// TwinCAT 3 PLC project SPS_Demo
// ProgramVersion: 3.1.4023.0
// libraries:
//   Tc2_ControllerToolbox, * (Beckhoff Automation GmbH)
//   Tc2_Math, * (Beckhoff Automation GmbH)
//   Tc2_MC2, * (Beckhoff Automation GmbH)
//   Tc2_MC2_Camming, * (Beckhoff Automation GmbH)
//   Tc2_Standard, * (Beckhoff Automation GmbH)
//   Tc2_System, * (Beckhoff Automation GmbH)
//   Tc2_Utilities, * (Beckhoff Automation GmbH)
//   Tc3_Module, * (Beckhoff Automation GmbH)
// project tree:
//   / AbwicklerTask.TcTTO, AufwicklerTask.TcTTO, DatenbearbeitungTask.TcTTO, FadenzugmotorTask.TcTTO, GlobalTextList.TcGTLO, MasterachseTask.TcTTO, PlcTask.TcTTO, Visualisierungsmanager.TcVMO (not stored)
//   DUTs/ DANCERCONTROL_ERRORS.TcDUT (not stored), DANCER_REF.TcDUT, E_DancerControlState.TcDUT (not stored), MoveState_t.TcDUT (not stored), MoveState_Fadenzugmotor.TcDUT (not stored), Regelungsmethode.TcDUT
//   GVLs/ GlobaleVariablen.TcGVL
//   POUs/Achsenzustandautom/ AbwicklerAnAus.TcPOU (not stored), AufwicklerAnAus.TcPOU, FadenzugmotorAnAus.TcPOU, MasterAnAus.TcPOU (not stored)
//   POUs/ MAIN.TcPOU
//   POUs/Regelungsmethode/ADRC-Regler/ ESO.TcPOU, Fal.TcPOU, TrackingDifferentiator.TcPOU, DiscreteTrackingDifferentiator.TcPOU, Sign.TcPOU
//   POUs/Regelungsmethode/IterativeLerningControl/ ILC.TcPOU, PRG_MovingAverage_1.TcPOU, Speicher_leeren.TcPOU
//   POUs/Regelungsmethode/KraftwerteBearbeiten/ Datenbearbeiten.TcPOU, PRG_Amplitudenbegrenzung.TcPOU, PRG_Analog2Volt.TcPOU, PRG_AntiPulsFilter.TcPOU, PRG_Durchschnitt.TcPOU, PRG_KalmannFilter.TcPOU, PRG_MovingAverage.TcPOU, PRG_Volt2Kraft.TcPOU
//   POUs/Regelungsmethode/PID-Regler/ PRG_PID_Abwickler.TcPOU, PRG_PID_Fadenzugmotor.TcPOU

CONFIGURATION SPS_Demo
    RESOURCE PLC ON TwinCAT3
        TASK AbwicklerTask(INTERVAL := T#100us, PRIORITY := 15);
        TASK AufwicklerTask(INTERVAL := T#100us, PRIORITY := 14);
        TASK DatenbearbeitungTask(INTERVAL := T#100us, PRIORITY := 2);
        TASK FadenzugmotorTask(INTERVAL := T#100us, PRIORITY := 3);
        TASK MasterachseTask(INTERVAL := T#100us, PRIORITY := 12);
        TASK PlcTask(INTERVAL := T#100us, PRIORITY := 1);
        PROGRAM AbwicklerAnAus WITH AbwicklerTask : AbwicklerAnAus;
        PROGRAM AufwicklerAnAus WITH AufwicklerTask : AufwicklerAnAus;
        PROGRAM Datenbearbeiten WITH DatenbearbeitungTask : Datenbearbeiten;
        PROGRAM Speicher_leeren WITH DatenbearbeitungTask : Speicher_leeren;
        PROGRAM FadenzugmotorAnAus WITH FadenzugmotorTask : FadenzugmotorAnAus;
        PROGRAM MasterAnAus WITH MasterachseTask : MasterAnAus;
        PROGRAM MAIN WITH PlcTask : MAIN;
    END_RESOURCE
END_CONFIGURATION

// ---- DUTs/DANCER_REF.TcDUT
TYPE DANCER_REF :
STRUCT
	/// 	Tension_ctl is the target value for web tension,
	///		typically the target position for the dancer in balanced condition 
	///	
	Tension_ctl: DINT;
	
	
	///	OUTPUT GearRatio
	///		GearRatio is the ratio of gear factor g(t)
	///		between master (web) and Slave (spool)
	///		to balance the dancer. Default is 1.0.
	///		GearRatio is an output value of the Dancercontrol function block.
	///	
	GearRatio: LREAL;
	
	
	
	/// 	deltaGear is the scaling multiplier of PID output (-1.0 ...  +1.0) to GearRatio - must be smaller than 1 but never 0.
	///		deltaGear would be e.g. 0.8 or 0.9 to limit the gear distortion 
	///		GearRatio = g(t) = deltaGear * PIDout + Gearoffset
	///	
	deltaGear: LREAL;
	
	
	
	/// 	GearOffset is the scaling offset to fit GearRatio distortion by satisfying equation
	///		GearRatio = g(t) = deltaGear * PIDout + Gearoffset
	///	
	GearOffset: LREAL;
	
	
	/// PID Control Proportional gain (P) 
	fKp: LREAL;
	
	
	/// PID Control Integral gain Tn (I) [s] 
	fTn: LREAL;
	
	
	/// PID Control Derivative gain Tv (D-T1) [s] 
	fTv: LREAL;
	
	
	/// PID Control Derivative damping time Td (D-T1) [s] 
	fTd: LREAL;
	
	
	/// 	acceleration limitation
	///		Accel_limit corresponds indirectly, i.e. relative to a
	///		maximum master velocity and to a maximum permitted 
	///		acceleration (pa = aSlaveMax / v MasterMax ). 
	///		The limit parameter pa corresponds to the 
	///		reciprocal value of the run-up time tH = 1 / pa 
	///	
	Accel_limit: LREAL;
END_STRUCT
END_TYPE

// ---- DUTs/Regelungsmethode.TcDUT
TYPE Regelungsmethode :
(
	Kraftkreis,
	On_Off
	
	
);
END_TYPE

// ---- GVLs/GlobaleVariablen.TcGVL
VAR_GLOBAL
	Master: 			AXIS_REF;
	Aufwickler: 		AXIS_REF;
	Abwickler: 			AXIS_REF;
	Fadenzugmotor		: AXIS_REF;		// Antrieb des Tänzers / Fadenzugausgleichssysmtems
	// Analog Input of EL3702 (Sample 0 ~ Sample 9 of Channel 1)
	aAnalogSamples_1 AT %I*: ARRAY[0..9] OF INT;
	// Analog Input of EL3702 (Sample 0 ~ Sample 9 of Channel 2)
	aAnalogSamples_2 AT %I*: ARRAY[0..9] OF INT;
	aAnalogSamplesReal_1: ARRAY[0..9] OF LREAL;
	aAnalogSamplesReal_2: ARRAY[0..9] OF LREAL;
	iAnalogSamplesAverageValue_1: LREAL := 0.36;
	iAnalogSamplesAverageValue_2: LREAL := 0.45;
	Reglerausgaenge: LREAL;
	ErrorTerm: LREAL;
	// Einheit (N)
	Sollkraft: LREAL := 10;
	Signal: LREAL;
	bPID_Regler_Switch: BOOL := FALSE;
	P_Regler_PseudoTorqCtrl_Out: LREAL;
	P_Regler_PTCVelocity_Out: LREAL;
	D_ReglerOut: LREAL;
	bI_Regler_Switch: BOOL := FALSE;
	bD_Regler_Switch: BOOL := FALSE;
	Fadenzugkraft_1: LREAL;
	Fadenzugkraft_2: LREAL;
	Sollposition: LREAL := 0;
	Istposition: LREAL;
	Stoerung: LREAL := 0;
	Stoerung_1: LREAL := 0;
	Stoerung_2: LREAL := 0;
	Positionsfehler: LREAL;
	KraftfehlerInPerzent: LREAL;
	stateAufwickler: Movestate_t;
	stateAbwickler: Movestate_t;
	xPunkt: LREAL := 360;
	MasterStart: BOOL;
	AufwicklerStart: BOOL;
	AbwicklerStart: BOOL;
	FadenmotorFreigabe: BOOL;
	MasterLaeuft: BOOL;
	AbwicklerLaeuft: BOOL;
	FadenzugHomingFertig: BOOL;
	FadenzugmotorLaeuft: BOOL;
	AufwicklerLaeuft: BOOL;
	Abwicklerstopp: BOOL;
	Aufwicklerstopp: BOOL;
	MasterStopp: BOOL;
	Straffunktion: LREAL;
	
	FadenmotorRegeln: BOOL:=FALSE;
	
	AbUndAufwicklersPosiabweichung: LREAL;
	AufwicklerJogStart: BOOL;
	FadenzugJogStart: BOOL;
	FadenzugmotorStopp: BOOL;
	NOT_AUS: BOOL;
	FadenzugmotorJogLaeuft: BOOL;
	AufwicklerJoglaeuft: BOOL;
	FadenzugmotorJogGes: LREAL;
	AufwicklerJogGes: LREAL;
	GearRatio: LREAL := 1;
	Regelungsmethode: STRING;
	v1: LREAL;
	v2: LREAL;
	ee:LREAL;//误差
	x1_hat:LREAL;//跟踪反馈值
	x2_hat:LREAL;//跟踪反馈值的而微分
	x3_hat:LREAL;//跟踪系统的扰动（总扰动）
	_u:LREAL;//输出值
	_u_neu: LREAL;
	u0:LREAL;//非线性组合系统输出
	
	ADRC_TD_r0:LREAL:=9000;
	ADRC_TD_h0:LREAL:=0.0001;
	// 3*wo
	ADRC_ESO_beta01:LREAL:=170;
	// 3*(wo^2)
	ADRC_ESO_beta02:LREAL:=5;
	// wo^3
	ADRC_ESO_beta03:LREAL:=0.01;
	b0:LREAL:=1.3;// 扰动补偿
	Referenzposition: LREAL := 90;
	ControlCycleTime: LREAL;
	P_Regler_Out_Abwickler: LREAL;
	I_Regler_Out_Abwickler: LREAL;
	I_Regler_Input_Abwickler: LREAL;
	D_Regler_Out_Abwickler: LREAL;
	PID_Output_After_Saturation_Abwickler: LREAL;
	//Kraftfehler: LREAL;
	PID_Output_After_Saturation_Fadenzugmotor: LREAL;
	Regler_Out_Fadenzugmotor: LREAL;
	P_Regler_Out_Fadenzugmotor: LREAL;
	I_Regler_Out_Fadenzugmotor: LREAL;
	D_Regler_Out_Fadenzugmotor: LREAL;
	I_Regler_Input_Fadenzugmotor: LREAL;
	// Grad
	MaxPosition: LREAL := 165;
	// Grad
	MinPosition: LREAL := 15;
	ADRC_Output:LREAL;
	KraftSensorNewValue: LREAL;
	KraftSensorOldValue: LREAL;
	Vorsteuerungsausgabe: LREAL;
	Kraftfehler: LREAL;
	KraftreglerOutput: LREAL;
	PID_Output_Old: ARRAY[0..20000] OF LREAL;
	ILC_Out: LREAL;
	k: INT := 2;
	Drehzahl: LREAL;
	u_new: LREAL;
	ILC_F_Out: LREAL;
	i:LREAL;
	LernenFertig: BOOL;
	ILC_EinAus:BOOL;
	neu_xPunkt: LREAL;
	alt_xPunkt: LREAL := xPunkt;
	xPunkt_geaendert: BOOL;
	u_Old: ARRAY[0..20000] OF LREAL;
	e_Old: ARRAY[0..20000] OF LREAL;
	count: INT;
	fla:BOOL:=FALSE;
	ADRC_ESO_h: LREAL := 0.0001;
	TD_Switch: BOOL;
	DTD_CTD: BOOL;
	E_Switch: BOOL;
END_VAR

// ---- POUs/Achsenzustandautom/AufwicklerAnAus.TcPOU
(* Ansteuerprogramm der Leitachse. Das Programm hat die Aufgabe, 
   die Leitachse in eine Bewegung konstanter Ge-schwindigkeit zu versetzen, 
   wieder anzuhalten und im Falle eines Fehlers die Achse durch einen Reset 
   wieder in einen funktionstüchtigen Zustand zu versetzen. *)

PROGRAM AufwicklerAnAus
VAR
	//stateMaster				: MoveState_t;		// Programmablauf über Zustandsvariable

	PowerAufwickler				: MC_Power;			// Schaltet Software-Freigabe der Leitachse
	HomeAufwicklerOut: ST_McOutputs;
	PowerAufwicklerOut			: ST_McOutputs;		// 
	
	ResetAufwickler				: MC_Reset;			// Setzt Achsfehler zurück
	ResetAufwicklerOut			: ST_McOutputs;	
	
	MoveAufwickler 				: MC_MoveVelocity;	// Versetzt Leitachse in Bewegung konstanter Geschwindigkeit
	MoveAufwicklerOut			: ST_McOutputs;
	
	HaltAufwickler				: MC_Halt;			// Hält Leitachse an
	GearInAufwicklerOut: ST_McOutputs;
	HaltAufwicklerOut			: ST_McOutputs;
	startAufwicklerTrig: R_TRIG;
	HaltAufwicklerTrig: R_TRIG;
	GearInAufwickler: MC_GearIn;
	GearOutAufwickler: MC_GearOut;
	CamOutAufwicklerOut: ST_McOutputs;
	CamInAufwicklerOut: ST_McOutputs;
	GearOutAufwicklerOut: ST_McOutputs;
	CamInAufwickler: MC_CamIn;
	CamOutAufwickler: MC_CamOut;
	SetCamOnlineChangeMode		: MC_SetCamOnlineChangeMode;				// Legt fest, wann und wie geänderte Kurvenscheibendaten übernommen werden
	SetCamOnlineChangeModeOut	: ST_McOutputs;
	
	CamTableSelect				: MC_CamTableSelect; // Spezifiziert und lädt Kurvenscheibentabelle in die NC
	
	MotionFunction				: ARRAY[1..4] OF MC_MotionFunctionPoint;	// Kurvenscheibe als Motion Function: Eindimensionale Liste (Array) von Stützstellen
	CamTable					: MC_CAM_REF;								// Referenz auf Kurvenscheibe: Beschreibung der Motion Function
	PointID						: MC_MotionFunctionPoint_ID;				// Wird den einzelnen Punkten/Stützstellen der Motion Function zugeordnet
	
	CamInfo						: MC_CamInfo;
	JogAufwicklerOut: ST_McOutputs;
	CamInfoOut					: ST_McOutputs;		
	CamInfoData					: MC_CamInfoData;	
	
	
	JogAufwickler: MC_Jog;
	flag: BOOL;
	AufwicklerHalt: MC_Halt;
	AufwicklerHaltOut: ST_McOutputs;
	HomeAufwickler: MC_Home;
	Kuppelungsmethode: BOOL;
	MARK: INT;
END_VAR

//startAufwicklerTrig(clk := MaschineStart);
//HaltAufwicklerTrig(clk := Abwicklerstopp);

GlobaleVariablen.Aufwickler();
CASE stateAufwickler OF
	
(* ===========================================================================================
   Zustand 1: Programm ist im Ausgangszustand und wartet auf Benutzereingabe. Alle 
   Funktionsbausteine werden initialisiert, etwaige Fehler zurückgesetzt. *)
	MOVESTATE_INIT :

		ResetAufwickler.Execute := FALSE;
		HaltAufwickler.Execute := FALSE;
		PowerAufwickler.Enable := FALSE;
		CamTableSelect.Execute := FALSE;
		CamInAufwickler.Execute := FALSE;
		CamOutAufwickler.Execute := FALSE;
		IF PowerAufwicklerOut.Active THEN
			ResetAufwickler.Execute := TRUE;
			IF ResetAufwickler.Done THEN
				AufwicklerLaeuft := FALSE;
				stateAufwickler := MOVESTATE_INIT;
			END_IF
		END_IF
		//HaltSlave.Execute := FALSE;
		//WriteMotionFunctionPoint.Execute := FALSE;
		//SetCamOnlineChangeMode.ActivationMode := MC_CAMACTIVATION_NEXTCYCLE;
		//SetCamOnlineChangeMode.MasterScalingMode := MC_CAMSCALING_AUTOOFFSET;
		//SetCamOnlineChangeMode.SlaveScalingMode := MC_CAMSCALING_AUTOOFFSET;
		IF AufwicklerStart = TRUE AND MasterLaeuft = FALSE THEN
			stateAufwickler := MOVESTATE_ENABLE;
		ELSIF AufwicklerStart = TRUE AND MasterLaeuft = TRUE THEN
			MasterStopp := TRUE;
		END_IF

(* ===========================================================================================
   Zustand 2: Schlalten der allgemeinen Software-Freigabe, Vorschubfreigabe in positive Richtung
   durch MC_Power. Sobald Funktionsbaustein MC_Power die Betriebsbereitschaft der Achse signalisiert,
   Zustandsübergang in Forward*)
	MOVESTATE_ENABLE :
			PowerAufwickler.Enable := TRUE;
			IF PowerAufwicklerOut.Done THEN
				stateAufwickler := MOVESTATE_HOMING;
			ELSIF PowerAufwickler.Error THEN
				stateAufwickler := MOVESTATE_ERROR;
			END_IF
	MOVESTATE_HOMING:
		IF AufwicklerStart = TRUE AND AufwicklerStopp = FALSE THEN
			HomeAufwickler.Execute := TRUE;

			IF HomeAufwicklerOut.Done THEN
				HomeAufwickler.Execute := FALSE;
				stateAufwickler := MOVESTATE_WRITEMOTIONFUNCTION;
				
			ELSIF HomeAufwicklerOut.CommandAborted OR HomeAufwicklerOut.Error THEN
				stateAufwickler := MOVESTATE_ERROR;
			END_IF
		END_IF	
(* ===========================================================================================
   Zustand 7: Beschreiben der zwei eindimensionalen Arrays mit der Stützstellen der Motion Function. 
   *)	
	MOVESTATE_WRITEMOTIONFUNCTION :
		PointID := 1;												// Dient nur der richtigen Position im Array
			MotionFunction[PointID].PointIndex			:= 1;		// Index der Stützstelle innerhalb der Motion Function
			MotionFunction[PointID].FunctionType 		:= 23;		// Modifizierte Sinuslinie
			MotionFunction[PointID].PointType    		:= 16#0002; // Motion Point Type : Rastpunkt
			MotionFunction[PointID].RelIndexNextPoint 	:= 1;		// Angabe des nächsten Punktes
			MotionFunction[PointID].MasterPos         	:= 0;		// x
			MotionFunction[PointID].SlavePos          	:= 0; 		// psi 
			MotionFunction[PointID].SlaveVelo         	:= 1; 		// psi'
			MotionFunction[PointID].SlaveAcc          	:= 0; 		// psi''
			MotionFunction[PointID].SlaveJerk         	:= 0; 		// psi'''
		
		PointID := 2;
			MotionFunction[PointID].PointIndex			:= 2;		// Polynom 1. Grades -> Gerade in Rast
			MotionFunction[PointID].FunctionType 		:= 23;
			MotionFunction[PointID].PointType    		:= 16#0002;
			MotionFunction[PointID].RelIndexNextPoint 	:= 1;
			MotionFunction[PointID].MasterPos         	:= 120;  	// x
			MotionFunction[PointID].SlavePos          	:= 180;  	// psi 
			MotionFunction[PointID].SlaveVelo         	:= 1; 		// psi'
			MotionFunction[PointID].SlaveAcc          	:= 0; 		// psi''
			MotionFunction[PointID].SlaveJerk         	:= 0; 		// psi'''
			
		PointID := 3;
			MotionFunction[PointID].PointIndex			:= 3;
			MotionFunction[PointID].FunctionType 		:= 23;
			MotionFunction[PointID].PointType    		:= 16#0002;
			MotionFunction[PointID].RelIndexNextPoint 	:= 1;   	// 
			MotionFunction[PointID].MasterPos         	:= 240;		// x
			MotionFunction[PointID].SlavePos          	:= 180;  	// psi 
			MotionFunction[PointID].SlaveVelo         	:= 1;   	// psi'
			MotionFunction[PointID].SlaveAcc          	:= 0; 		// psi''
			MotionFunction[PointID].SlaveJerk         	:= 0; 		// psi'''
			
			
		PointID := 4;
			MotionFunction[PointID].PointIndex			:= 4;
			MotionFunction[PointID].FunctionType 		:= 23;
			MotionFunction[PointID].PointType    		:= 16#0002;
			MotionFunction[PointID].RelIndexNextPoint 	:= 0;   	// 0, da es keinen nächsten Punkt gibt
			MotionFunction[PointID].MasterPos         	:= 360;		// x
			MotionFunction[PointID].SlavePos          	:= 360;  	// psi 
			MotionFunction[PointID].SlaveVelo         	:= 1;   	// psi'
			MotionFunction[PointID].SlaveAcc          	:= 0; 		// psi''
			MotionFunction[PointID].SlaveJerk         	:= 0; 		// psi'''

(*
		PointID := 5;
			MotionFunction[PointID].PointIndex			:= 5;
			MotionFunction[PointID].FunctionType 		:= 1;
			MotionFunction[PointID].PointType    		:= 16#0001;
			MotionFunction[PointID].RelIndexNextPoint 	:= 0;   	// 0, da es keinen nächsten Punkt gibt
			MotionFunction[PointID].MasterPos         	:= x5;		// x
			MotionFunction[PointID].SlavePos          	:= 360;  	// psi 
			MotionFunction[PointID].SlaveVelo         	:= 1;   	// psi'
			MotionFunction[PointID].SlaveAcc          	:= 0; 		// psi''
			MotionFunction[PointID].SlaveJerk         	:= 0; 		// psi'''
			*)
		stateAufwickler := MOVESTATE_CAMTABLESELECT;		
		
		
	(* ===========================================================================================
   Zustand 8: Einlesen, Spezifizieren und in die NC laden der Kurvenscheibendaten. 
   Erste Kurvenscheibe *)	
	MOVESTATE_CAMTABLESELECT :
	
		CamInAufwickler.CamTableID := 1;										 // Festlegung der Kurvenscheiben-ID
		CamTable.TableType := MC_TABLETYPE_MOTIONFUNCTION; 						 // Motion Function und keine Positionstabelle
		CamTable.pArray := ADR(MotionFunction);									 // Adresse des Arrays, der die Stützstellen hält
		CamTable.ArraySize := SIZEOF(MotionFunction);							 // Speichergröße des Arrays
		CamTable.NoOfColumns := 1;												 // Spaltenzahl 
		CamTable.NoOfRows := SIZEOF(MotionFunction) / SIZEOF(MotionFunction[1]); // Zeilenzahl: Gesamtspeicherplatz durch Speicherplatz einer Zeile
		CamTableSelect.Execute := TRUE;
		IF CamTableSelect.Done THEN
			CamTableSelect.Execute := FALSE;
			stateAufwickler := MOVESTATE_CAMIN;
		ELSIF CamTableSelect.Error THEN
			stateAufwickler := MOVESTATE_ERROR;
		END_IF	
		
	MOVESTATE_CAMIN :
		IF AufwicklerStart = TRUE AND AufwicklerStopp = FALSE THEN
			CamInAufwickler.CamTableID := 1;											// Kopplung  mit ID 1
			CamInAufwickler.MasterOffset := 0;										  	// Weder Offset...
			CamInAufwickler.SlaveOffset := 0;
			CamInAufwickler.MasterScaling := 1.0;										// ... noch Skalierung erforderlich
			CamInAufwickler.SlaveScaling := 1.0;
			CamInAufwickler.StartMode := MC_STARTMODE_RELATIVE;						  	// Ursprung des Kurvenscheibenkoordinatensystemes an akt. Achsposition
			CamInAufwickler.Execute := TRUE;
			IF CamInAufwickler.InSync THEN											  	// Kopplung erfolgreich, Kurvenscheibe aktiv
				CamInAufwickler.Execute := FALSE;
				stateAufwickler := MOVESTATE_FORWARD;
			ELSIF CamInAufwickler.CommandAborted OR CamInAufwickler.Error THEN
				stateAufwickler := MOVESTATE_ERROR;
			END_IF
		ELSIF AufwicklerStart = FALSE THEN
			stateAufwickler := MOVESTATE_STOPAUFWICKLER;
		END_IF
		
	MOVESTATE_FORWARD :
		
		IF AufwicklerStart = TRUE AND AufwicklerStopp = FALSE THEN
			AufwicklerLaeuft := TRUE;
			IF AufwicklerJogStart = TRUE THEN
				flag := TRUE;
				stateAufwickler := MOVESTATE_STOPAUFWICKLER;
			END_IF
			IF CamInAufwicklerOut.Done THEN
				AufwicklerLaeuft := TRUE;
			END_IF
		ELSE
			stateAufwickler := MOVESTATE_STOPAUFWICKLER;
		END_IF		

(* ===========================================================================================
   Zustand 4: Anhalten der Leitachse, im Anschluss Rückkehr in den Ausgangszustand. *)		
	MOVESTATE_STOPAUFWICKLER :
		CamOutAufwickler.Execute := TRUE;
		IF CamOutAufwicklerOut.Done THEN
			IF AufwicklerHaltOut.Done THEN	
				AufwicklerHalt.Execute := FALSE;
				IF flag = TRUE AND AufwicklerJogStart = TRUE THEN
					flag := FALSE;
					AufwicklerStopp := FALSE;
					AufwicklerStart := TRUE;
					stateAufwickler := MOVESTATE_JOG;
				ELSE
					AufwicklerStopp := TRUE;
					AufwicklerStart := FALSE;
					AufwicklerLaeuft := FALSE;
					stateAufwickler := MOVESTATE_INIT;
				END_IF
			ELSE
				AufwicklerHalt.Execute := TRUE;
			END_IF
			
			
		ELSIF CamOutAufwickler.Error THEN
			CamOutAufwickler.Execute := FALSE;
			stateAufwickler := MOVESTATE_ERROR;
		END_IF
		
	MOVESTATE_JOG:
		AufwicklerLaeuft := TRUE;
		AufwicklerJoglaeuft := TRUE;
		IF AufwicklerJogStart = FALSE THEN
			AufwicklerJoglaeuft := FALSE;
			stateAufwickler := MOVESTATE_INIT;
		END_IF
	
(* ===========================================================================================
   Zustand 5: Im Falle eines Bausteinfehlers wird überprüft, ob sich die Achse ebenfalls im    
   Fehlerzustand befindet, was einen Achsreset erfordert. Andernfalls werden Bausteinfehler 
   im Zustand Init zurückgesetzt.*)		
	MOVESTATE_ERROR :
		IF Master.Status.Error THEN
			stateAufwickler := MOVESTATE_RESET;	// Reset bei Achsfehler
		ELSE
			stateAufwickler := MOVESTATE_INIT;	// Funktionsbausteinfehler erfordert keinen Reset
		END_IF

(* ===========================================================================================
   Zustand 6:  Durchführung des Achsreset im Fehlerfall  *)		
	MOVESTATE_RESET :
		CamInAufwickler.Execute := FALSE;
		ResetAufwickler.Execute := TRUE;
		IF ResetAufwickler.Done THEN
			AufwicklerLaeuft := FALSE;
			stateAufwickler := MOVESTATE_INIT;
		ELSIF ResetAufwickler.Error THEN
			stateAufwickler := MOVESTATE_INIT; (* Falls Reset nicht gelingt, Benutzereingriff erforderlich *)
		END_IF
		
END_CASE

// Zyklusmäßige Aufrufe
ActPower();		// Aufruf des Power Funktionsbausteines
ActCamming();	// Aufruf des Camming-Funktionsbausteines
ActReset();		// Aufruf des Reset-Funktionsbausteines
ActJog();
ActHalt();
ActHome();

ACTION ActCamming:
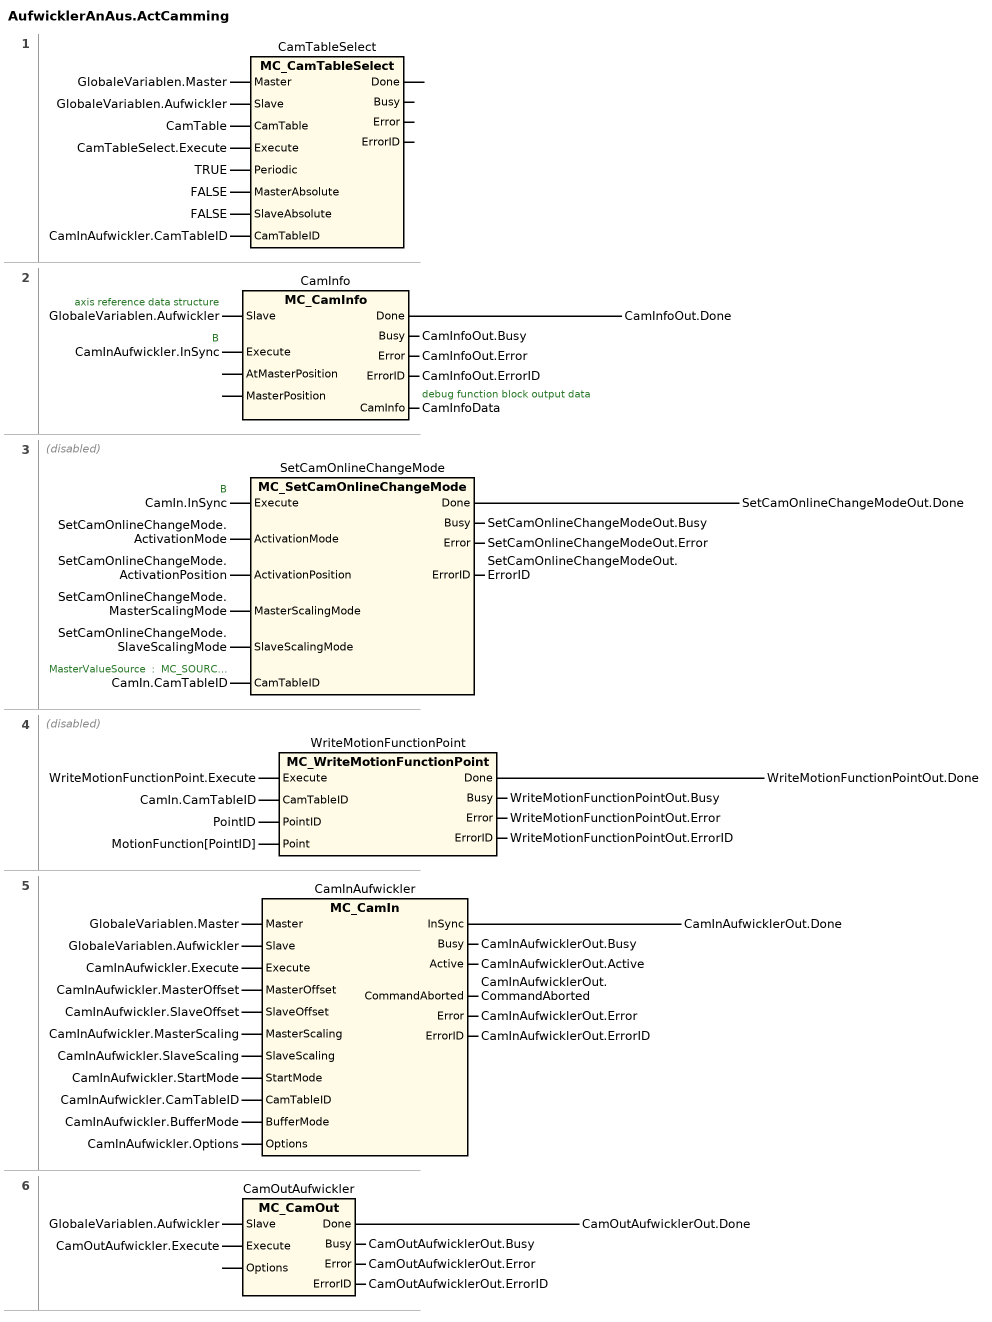
// NETWORK 1
CamTableSelect(
    Master := GlobaleVariablen.Master,
    Slave := GlobaleVariablen.Aufwickler,
    CamTable := CamTable,
    Execute := CamTableSelect.Execute,
    Periodic := TRUE,
    MasterAbsolute := FALSE,
    SlaveAbsolute := FALSE,
    CamTableID := CamInAufwickler.CamTableID); // MC_CamTableSelect

// NETWORK 2
//   GlobaleVariablen.Aufwickler: axis reference data structure
//   CamInAufwickler.InSync: B
//   CamInfoData: debug function block output data
CamInfo(
    Slave := GlobaleVariablen.Aufwickler,
    Execute := CamInAufwickler.InSync,
    Busy => CamInfoOut.Busy,
    Error => CamInfoOut.Error,
    ErrorID => CamInfoOut.ErrorID,
    CamInfo => CamInfoData); // MC_CamInfo
CamInfoOut.Done := CamInfo.Done;

// NETWORK 3 (disabled)
//   CamIn.InSync: B
//   CamIn.CamTableID: MasterValueSource : MC_SOURCE E not available
// SetCamOnlineChangeMode(
//     Execute := CamIn.InSync,
//     ActivationMode := SetCamOnlineChangeMode.ActivationMode,
//     ActivationPosition := SetCamOnlineChangeMode.ActivationPosition,
//     MasterScalingMode := SetCamOnlineChangeMode.MasterScalingMode,
//     SlaveScalingMode := SetCamOnlineChangeMode.SlaveScalingMode,
//     CamTableID := CamIn.CamTableID,
//     Busy => SetCamOnlineChangeModeOut.Busy,
//     Error => SetCamOnlineChangeModeOut.Error,
//     ErrorID => SetCamOnlineChangeModeOut.ErrorID); // MC_SetCamOnlineChangeMode
// SetCamOnlineChangeModeOut.Done := SetCamOnlineChangeMode.Done;

// NETWORK 4 (disabled)
// WriteMotionFunctionPoint(
//     Execute := WriteMotionFunctionPoint.Execute,
//     CamTableID := CamIn.CamTableID,
//     PointID := PointID,
//     Point := MotionFunction[PointID],
//     Busy => WriteMotionFunctionPointOut.Busy,
//     Error => WriteMotionFunctionPointOut.Error,
//     ErrorID => WriteMotionFunctionPointOut.ErrorID); // MC_WriteMotionFunctionPoint
// WriteMotionFunctionPointOut.Done := WriteMotionFunctionPoint.Done;

// NETWORK 5
CamInAufwickler(
    Master := GlobaleVariablen.Master,
    Slave := GlobaleVariablen.Aufwickler,
    Execute := CamInAufwickler.Execute,
    MasterOffset := CamInAufwickler.MasterOffset,
    SlaveOffset := CamInAufwickler.SlaveOffset,
    MasterScaling := CamInAufwickler.MasterScaling,
    SlaveScaling := CamInAufwickler.SlaveScaling,
    StartMode := CamInAufwickler.StartMode,
    CamTableID := CamInAufwickler.CamTableID,
    BufferMode := CamInAufwickler.BufferMode,
    Options := CamInAufwickler.Options,
    Busy => CamInAufwicklerOut.Busy,
    Active => CamInAufwicklerOut.Active,
    CommandAborted => CamInAufwicklerOut.CommandAborted,
    Error => CamInAufwicklerOut.Error,
    ErrorID => CamInAufwicklerOut.ErrorID); // MC_CamIn
CamInAufwicklerOut.Done := CamInAufwickler.InSync;

// NETWORK 6
CamOutAufwickler(
    Slave := GlobaleVariablen.Aufwickler,
    Execute := CamOutAufwickler.Execute,
    Busy => CamOutAufwicklerOut.Busy,
    Error => CamOutAufwicklerOut.Error,
    ErrorID => CamOutAufwicklerOut.ErrorID); // MC_CamOut
CamOutAufwicklerOut.Done := CamOutAufwickler.Done;
END_ACTION

ACTION ActGearInDyn:
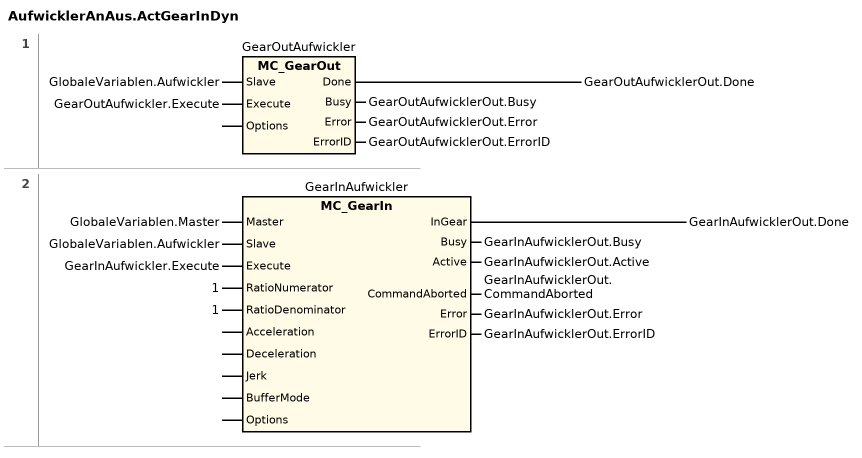
// NETWORK 1
GearOutAufwickler(
    Slave := GlobaleVariablen.Aufwickler,
    Execute := GearOutAufwickler.Execute,
    Busy => GearOutAufwicklerOut.Busy,
    Error => GearOutAufwicklerOut.Error,
    ErrorID => GearOutAufwicklerOut.ErrorID); // MC_GearOut
GearOutAufwicklerOut.Done := GearOutAufwickler.Done;

// NETWORK 2
GearInAufwickler(
    Master := GlobaleVariablen.Master,
    Slave := GlobaleVariablen.Aufwickler,
    Execute := GearInAufwickler.Execute,
    RatioNumerator := 1,
    RatioDenominator := 1,
    Busy => GearInAufwicklerOut.Busy,
    Active => GearInAufwicklerOut.Active,
    CommandAborted => GearInAufwicklerOut.CommandAborted,
    Error => GearInAufwicklerOut.Error,
    ErrorID => GearInAufwicklerOut.ErrorID); // MC_GearIn
GearInAufwicklerOut.Done := GearInAufwickler.InGear;
END_ACTION

ACTION ActHalt:
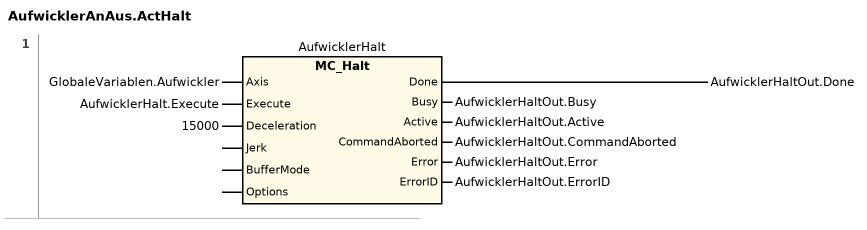
// NETWORK 1
AufwicklerHalt(
    Axis := GlobaleVariablen.Aufwickler,
    Execute := AufwicklerHalt.Execute,
    Deceleration := 15000,
    Busy => AufwicklerHaltOut.Busy,
    Active => AufwicklerHaltOut.Active,
    CommandAborted => AufwicklerHaltOut.CommandAborted,
    Error => AufwicklerHaltOut.Error,
    ErrorID => AufwicklerHaltOut.ErrorID); // MC_Halt
AufwicklerHaltOut.Done := AufwicklerHalt.Done;
END_ACTION

ACTION ActHome:
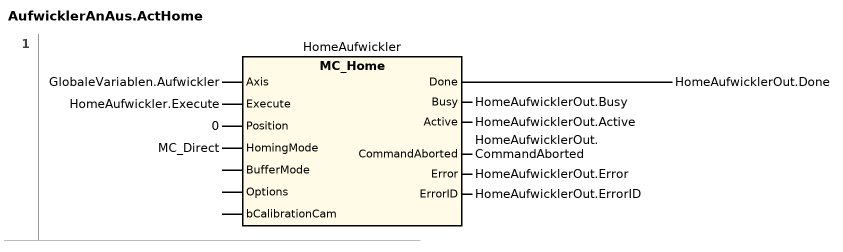
// NETWORK 1
HomeAufwickler(
    Axis := GlobaleVariablen.Aufwickler,
    Execute := HomeAufwickler.Execute,
    Position := 0,
    HomingMode := MC_Direct,
    Busy => HomeAufwicklerOut.Busy,
    Active => HomeAufwicklerOut.Active,
    CommandAborted => HomeAufwicklerOut.CommandAborted,
    Error => HomeAufwicklerOut.Error,
    ErrorID => HomeAufwicklerOut.ErrorID); // MC_Home
HomeAufwicklerOut.Done := HomeAufwickler.Done;
END_ACTION

ACTION ActJog:
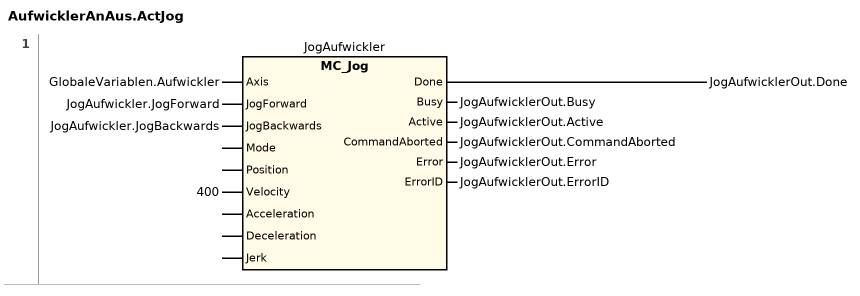
// NETWORK 1
JogAufwickler(
    Axis := GlobaleVariablen.Aufwickler,
    JogForward := JogAufwickler.JogForward,
    JogBackwards := JogAufwickler.JogBackwards,
    Velocity := 400,
    Busy => JogAufwicklerOut.Busy,
    Active => JogAufwicklerOut.Active,
    CommandAborted => JogAufwicklerOut.CommandAborted,
    Error => JogAufwicklerOut.Error,
    ErrorID => JogAufwicklerOut.ErrorID); // MC_Jog
JogAufwicklerOut.Done := JogAufwickler.Done;
END_ACTION

ACTION ActPower:
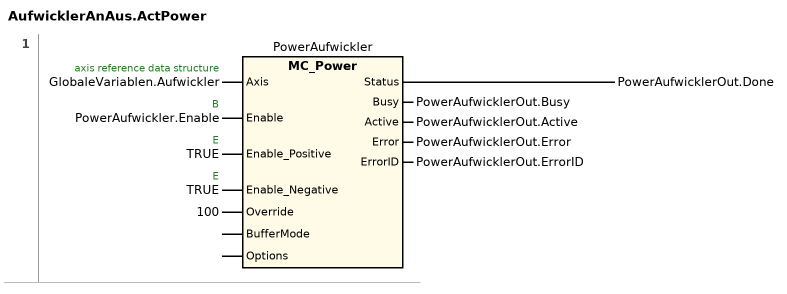
// NETWORK 1
//   GlobaleVariablen.Aufwickler: axis reference data structure
//   PowerAufwickler.Enable: B
//   TRUE: E
PowerAufwickler(
    Axis := GlobaleVariablen.Aufwickler,
    Enable := PowerAufwickler.Enable,
    Enable_Positive := TRUE,
    Enable_Negative := TRUE,
    Override := 100,
    Busy => PowerAufwicklerOut.Busy,
    Active => PowerAufwicklerOut.Active,
    Error => PowerAufwicklerOut.Error,
    ErrorID => PowerAufwicklerOut.ErrorID); // MC_Power
PowerAufwicklerOut.Done := PowerAufwickler.Status;
END_ACTION

ACTION ActReset:
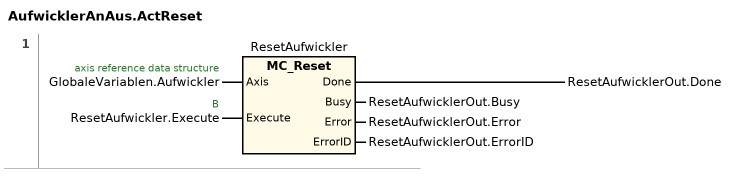
// NETWORK 1
//   GlobaleVariablen.Aufwickler: axis reference data structure
//   ResetAufwickler.Execute: B
ResetAufwickler(
    Axis := GlobaleVariablen.Aufwickler,
    Execute := ResetAufwickler.Execute,
    Busy => ResetAufwicklerOut.Busy,
    Error => ResetAufwicklerOut.Error,
    ErrorID => ResetAufwicklerOut.ErrorID); // MC_Reset
ResetAufwicklerOut.Done := ResetAufwickler.Done;
END_ACTION

END_PROGRAM

// ---- POUs/Regelungsmethode/KraftwerteBearbeiten/Datenbearbeiten.TcPOU
PROGRAM Datenbearbeiten
VAR
	bFilterSwitch: BOOL := TRUE;
END_VAR

// wenn der Fadenzugsensor eingeschaltet wird, ist der Anfangswert ca. 1500. 
IF GlobaleVariablen.aAnalogSamples_2[0]>999 THEN //um einfach festzustellen, ob der Sensor funktioniert
	
	PRG_Analog2Volt();			   // LREAL -> Volt(V):  0-32767 -> 0-10 V
	
	IF bFilterSwitch THEN          // Filter nutzen. Nachteil: Zeitverzögerung von mindestens einem Task-Zykluszeit(Bei diesem Programm ist die Zeitverzögerung gegen 0.1 ms)
		PRG_AntiPulsFilter();	   // die Höchst- und Mindestwerte aus der Proben entfernen und danach Durchschnitt ermitteln.
		PRG_Amplitudenbegrenzung();//der neue Wert entfernen, wenn der neue Wert 2 mal größer als der alte Wert.
		PRG_KalmannFilter();	   // Trendvorhersage und Rollendes Filtrieren
		//PRG_MovingAverage();      // Der Filter kommt aus Beckhoff
	ELSE						   // Filter nicht nutzen, aber unsere Analogklemme EL3702 gibt uns 10 Stichproben in jedem Task-Zyklus. 
		PRG_Durchschnitt();		   // die Mittelwert der 10 Stichproben ermittteln
	END_IF
	
	PRG_Volt2Kraft();			   // Volt(V) -> Kraft(N)
END_IF

END_PROGRAM

// ---- POUs/Regelungsmethode/KraftwerteBearbeiten/PRG_Analog2Volt.TcPOU
PROGRAM PRG_Analog2Volt
VAR
	i: INT;
END_VAR

FOR i := 0 TO 9 BY 1 DO
	//Eingangswerte sind 0-32767 (LREAL)
	IF GlobaleVariablen.aAnalogSamples_2[i] < 0 THEN
		GlobaleVariablen.aAnalogSamples_2[i] := 0;
	ELSIF GlobaleVariablen.aAnalogSamples_2[i] > 32767 THEN
		GlobaleVariablen.aAnalogSamples_2[i] := 32767;
	END_IF
	
	//LREAL -> Volt(V) 0-32767 -> 0-10 V
	GlobaleVariablen.aAnalogSamplesReal_2[i] := (10.0 / 32767.0) * GlobaleVariablen.aAnalogSamples_2[i]; // (0.000305185094759 = 10.0 / 32767.0)
	
END_FOR

END_PROGRAM

// ---- POUs/Regelungsmethode/KraftwerteBearbeiten/PRG_AntiPulsFilter.TcPOU
PROGRAM PRG_AntiPulsFilter
VAR
	i: INT;
	lmax_1: LREAL;
	lmax_2: LREAL;
	lmin_1: LREAL;
	lmin_2: LREAL;
	lsum_1: LREAL;
	lsum_2: LREAL;
END_VAR

//Anti-Puls-Interferenz-Filterverfahren
//die Höchst- und Mindestwerte aus der Proben entfernen und danach Durchschnitt ermitteln.
lsum_2 := 0;
lmax_2 := GlobaleVariablen.aAnalogSamplesReal_2[0];
lmin_2 := GlobaleVariablen.aAnalogSamplesReal_2[0];

FOR i := 0 TO 9 BY 1 DO
	IF lmax_2 < GlobaleVariablen.aAnalogSamplesReal_2[i] THEN
		lmax_2 := GlobaleVariablen.aAnalogSamplesReal_2[i];
	END_IF
	IF lmin_2 > GlobaleVariablen.aAnalogSamplesReal_2[i] THEN
		lmin_2 := GlobaleVariablen.aAnalogSamplesReal_2[i];
	END_IF
	lsum_2 := lsum_2 + GlobaleVariablen.aAnalogSamplesReal_2[i];
END_FOR

//GlobaleVariablen.iAnalogSamplesAverageValue := (isum-imax-imin)/8;
KraftSensorNewValue := (lsum_2 - lmax_2 - lmin_2) / 8;

END_PROGRAM

// ---- POUs/Regelungsmethode/KraftwerteBearbeiten/PRG_Amplitudenbegrenzung.TcPOU
PROGRAM PRG_Amplitudenbegrenzung
VAR
END_VAR

//*********************************
//Amplitudenbegrenzende Filterungsmethode
//der neue Wert entfernen, wenn der neue Wert 2 mal größer als der alte Wert.

IF (KraftSensorNewValue - GlobaleVariablen.iAnalogSamplesAverageValue_2 > 2) OR (GlobaleVariablen.iAnalogSamplesAverageValue_2 - KraftSensorNewValue> 2) THEN
	GlobaleVariablen.iAnalogSamplesAverageValue_2 := KraftSensorOldValue;
ELSE
	GlobaleVariablen.iAnalogSamplesAverageValue_2 := KraftSensorNewValue;
END_IF
KraftSensorOldValue := GlobaleVariablen.iAnalogSamplesAverageValue_2;
//*********************************

END_PROGRAM

// ---- POUs/Regelungsmethode/KraftwerteBearbeiten/PRG_KalmannFilter.TcPOU
PROGRAM PRG_KalmannFilter
VAR
	P: LREAL := 1.0;
	P_: LREAL;
	X: LREAL := 0.0;
	X_: LREAL;
	K: LREAL := 0;
	Q: LREAL := 0.001;
	// 1
	RR: LREAL := 0.1;
	OriginalOutput: LREAL;
END_VAR

//*********************************
//Kalmann Filter
OriginalOutput := GlobaleVariablen.iAnalogSamplesAverageValue_2;
X_ := X + 0;
P_ := P + Q;
K := P_ / (P_ + RR);
X := X_ + K * (GlobaleVariablen.iAnalogSamplesAverageValue_2 - X_);
P := P_ - K * P_;
GlobaleVariablen.iAnalogSamplesAverageValue_2 := X;
//*********************************

END_PROGRAM

// ---- POUs/Regelungsmethode/KraftwerteBearbeiten/PRG_Durchschnitt.TcPOU
PROGRAM PRG_Durchschnitt
VAR
END_VAR

GlobaleVariablen.iAnalogSamplesAverageValue_2 := (10.0 / 32767.0) * INT_TO_LREAL((GlobaleVariablen.aAnalogSamples_2[0] + 
																				 GlobaleVariablen.aAnalogSamples_2[1] +
																				 GlobaleVariablen.aAnalogSamples_2[2] +
																				 GlobaleVariablen.aAnalogSamples_2[3] +
																				 GlobaleVariablen.aAnalogSamples_2[4] +
																				 GlobaleVariablen.aAnalogSamples_2[5] +
																				 GlobaleVariablen.aAnalogSamples_2[6] +
																				 GlobaleVariablen.aAnalogSamples_2[7] +
																				 GlobaleVariablen.aAnalogSamples_2[8] +
																				 GlobaleVariablen.aAnalogSamples_2[9]) / 10); // (0.000305185094759 = 10.0 / 32767.0)

END_PROGRAM

// ---- POUs/Regelungsmethode/KraftwerteBearbeiten/PRG_Volt2Kraft.TcPOU
PROGRAM PRG_Volt2Kraft
VAR
END_VAR

//Volt(V) -> Kraft(N) 
IF GlobaleVariablen.iAnalogSamplesAverageValue_2 > 0.42 THEN // In der Sensoranleitung ist die Wert 0,5 -> 0,5 ist nicht richtig für diese Fadenzugsensor. 0,42 ist richtig.
	//Jeder Kraftsensor hat einen anderen Wert, für diesen Sensor muss der Ausgangswert um  0.40 oder 0.41 abgezogen werden.
	GlobaleVariablen.Fadenzugkraft_2 := 100 * ((GlobaleVariablen.iAnalogSamplesAverageValue_2 - 0.402)/4.0);// Die Formel kommt aus der Sensoranleitung, aber wie gesagt, dass 0,4 ist bei mir ausgewählt.
ELSE GlobaleVariablen.Fadenzugkraft_2 := 0;
END_IF

END_PROGRAM

// ---- POUs/Regelungsmethode/IterativeLerningControl/Speicher_leeren.TcPOU
PROGRAM Speicher_leeren
VAR
	m:INT;
END_VAR

IF xPunkt_geaendert = TRUE OR (ILC_EinAus = FALSE AND MasterStart = TRUE) THEN
	FOR m := 0 TO 2000 BY 1 DO
		u_Old[m]:= 0;
		e_Old[m]:= 0;
		count := 0;
	END_FOR
	LernenFertig := FALSE;
	ILC_Out := 0;
	alt_xPunkt := xPunkt;
END_IF

END_PROGRAM

// ---- POUs/Achsenzustandautom/FadenzugmotorAnAus.TcPOU
PROGRAM FadenzugmotorAnAus
VAR
	PowerFadenzugmotor: MC_Power;
	PowerFadenzugmotorOut: ST_McOutputs;
	ResetFadenzugmotor: MC_Reset;
	ResetFadenzugmotorOut: ST_McOutputs;
	HaltFadenzugmotor: MC_Halt;
	HaltFadenzugmotorOut: ST_McOutputs;
	HomeFadenzugmotor: MC_Home;
	HomeFadenzugmotorOut: ST_McOutputs;
	MoveAbFadenzugmotorOut1: ST_McOutputs;
	MoveAbFadenzugmotor1: MC_MoveAbsolute;
	MoveAbFadenzugmotor2: MC_MoveAbsolute;
	MoveAbFadenzugmotorOut2: ST_McOutputs;
	MC_Stop1: MC_Stop;
	MC_StopOut1: ST_McOutputs;
	HaltAufwicklerOut: ST_McOutputs;
	HaltAbwicklerOut: ST_McOutputs;
	AbwicklerMoveV_Out: ST_McOutputs;
	AufwicklerMoveV: MC_MoveVelocity;
	HaltAbwickler: MC_Halt;
	HaltAufwickler: MC_Halt;
	PowerAbwickler: MC_Power;
	PowerAbwicklerOut: ST_McOutputs;
	PowerAufwickler: MC_Power;
	PowerAufwicklerOut: ST_McOutputs;
	HomeAbwickler: MC_Home;
	HomeAbwicklerOut: ST_McOutputs;
	HomeAufwickler: MC_Home;
	HomeAufwicklerOut: ST_McOutputs;
	ResetAbwickler: MC_Reset;
	ResetAbwickleOUT: ST_McOutputs;
	ResetAufwickler: MC_Reset;
	ResetAufwickleOUT: ST_McOutputs;
	MasterMoveV: MC_MoveVelocity;
	HaltMasterachse: MC_Halt;
	ResetMasterachseOut: ST_McOutputs;
	HomeMasterachseOut: ST_McOutputs;
	HaltMasterachseOut: ST_McOutputs;
	PowerMasterachseOut: ST_McOutputs;
	GearIn_M_AB_Out: ST_McOutputs;
	MasterMoveV_Out: ST_McOutputs;
	PowerMasterachse: MC_Power;
	HomeMasterachse: MC_Home;
	ResetMasterachse: MC_Reset;
	GearIn_M_AB: MC_GearIn;
	GearOut_M_AB: MC_GearOut;
	CamIn_AB_AUF_Out: ST_McOutputs;
	GearOut_M_AB_Out: ST_McOutputs;
	CamIn_AB_AUF: MC_CamIn;
	CamOut_AB_AUF: MC_CamOut;
	JogFadenzugmotorOut: ST_McOutputs;
	CamOut_AB_AUF_Out: ST_McOutputs;
	startFadenzugTrig: R_TRIG;
	flag: INT;
	JogFadenzugmotor: MC_Jog;
	// Zustandsvariable Hauptprogramm
	stateFadenzugmotor: MoveState_Fadenzugmotor;
	
END_VAR

GlobaleVariablen.Fadenzugmotor();
IF Fadenzugmotor.NcToPlc.ActPos > 89 AND Fadenzugmotor.NcToPlc.ActPos < 91 THEN
	FadenzugHomingFertig := TRUE;
ELSE FadenzugHomingFertig := FALSE;
END_IF
IF DTD_CTD THEN
	TrackingDifferentiator(Sollkraft);
ELSE
	DiscreteTrackingDifferentiator(Sollkraft);
END_IF

ESO(Fadenzugkraft_2);

// Programmablauf mittels Zustandsautomat
CASE stateFadenzugmotor OF
(* ===========================================================================================
	Zustand 1: Programm ist im Ausgangszustand und wartet auf Benutzereingabe. Alle 
	Funktionsbausteine werden initialisiert, etwaige Fehler zurückgesetzt. *)	
	FADENZUG_INIT:
		FadenzugmotorStopp := FALSE;
		MoveAbFadenzugmotor1.Execute := FALSE;
		MoveAbFadenzugmotor2.Execute := FALSE;
		FadenzugmotorLaeuft := FALSE;
		ResetFadenzugmotor.Execute := FALSE;
		HaltFadenzugmotor.Execute := FALSE;
		FadenmotorRegeln := FALSE;
		IF FadenmotorFreigabe THEN
			stateFadenzugmotor := FADENZUG_POWER_ON;
		ELSE
			PowerFadenzugmotor.Enable := FALSE;
			PowerFadenzugmotor.Enable_Positive := FALSE;
			PowerFadenzugmotor.Enable_Negative := FALSE;
		END_IF
(* ===========================================================================================
	Zustand 2: Schlalten der allgemeinen Software-Freigabe, Vorschubfreigabe in positive Richtung
	durch MC_Power. Sobald Funktionsbaustein MC_Power die Betriebsbereitschaft der Achse signalisiert,
	Zustandsübergang in Forward*)
	FADENZUG_POWER_ON:
		IF FadenmotorFreigabe = TRUE THEN
			PowerFadenzugmotor.Enable := TRUE;
			PowerFadenzugmotor.Enable_Positive := TRUE;
			PowerFadenzugmotor.Enable_Negative := TRUE;
			FadenzugmotorStopp := FALSE;
			IF PowerFadenzugmotorOut.Done THEN
				IF FadenzugJogStart THEN
					stateFadenzugmotor := FADENZUG_JOG;
				END_IF
			ELSIF PowerFadenzugmotor.Error THEN
				stateFadenzugmotor := FADENZUG_ERROR;
			END_IF
		ELSIF FadenmotorFreigabe = FALSE THEN
			stateFadenzugmotor := FADENZUG_HALT_ZU_INT;
		END_IF
(* ===========================================================================================
	Zustand 3: Setzten der Ist-Position auf 90 Grad*)			
	FADENZUG_JOG:
		IF FadenmotorFreigabe = TRUE THEN
			FadenzugmotorJogLaeuft := TRUE;
			ActJog();
			IF FadenzugJogStart = FALSE THEN
				FadenzugmotorJogLaeuft := FALSE;
				IF FadenmotorRegeln = TRUE THEN
					stateFadenzugmotor := FADENZUG_MOVE;
				END_IF
			END_IF
		ELSIF FadenmotorFreigabe = FALSE THEN
			stateFadenzugmotor := FADENZUG_HALT_ZU_INT;
		END_IF
(* ===========================================================================================
	Zustand 4: Starten des Fadenzugmotors mithilfe der Fadenzugspannung. Zustandsübergang durch Bedienerbefehl.*)	
	FADENZUG_MOVE:
	
		IF FadenmotorFreigabe = TRUE THEN
			
			IF FadenzugmotorStopp = TRUE THEN
				FadenmotorFreigabe := FALSE;
			END_IF
			//*********Positionsführungsgröße berechnen*************
			PRG_PID_Fadenzugmotor();
			IF ILC_EinAus = TRUE AND MasterStart = TRUE THEN
				ILC();
				MoveAbFadenzugmotor1.Position := ILC_Out + GlobaleVariablen.Fadenzugmotor.NcToPlc.ActPos + _u;
			ELSE
				MoveAbFadenzugmotor1.Position := GlobaleVariablen.Fadenzugmotor.NcToPlc.ActPos + _u;
			END_IF
			
			MoveAbFadenzugmotor1.Velocity := 60000;
			ActBegrenzung_1();
			//******************************************************
			
			MoveAbFadenzugmotor1.Execute := TRUE;
			FadenzugmotorLaeuft := TRUE;
			
			//*********Zustand umschalten***************************
			IF MoveAbFadenzugmotorOut1.Busy OR MoveAbFadenzugmotorOut1.Active THEN
				MoveAbFadenzugmotor1.Execute := FALSE;
				stateFadenzugmotor := FADENZUG_MOVE_NEW;
			END_IF
			
			IF MoveAbFadenzugmotorOut1.Done OR MoveAbFadenzugmotorOut1.CommandAborted THEN
				MoveAbFadenzugmotor1.Execute := FALSE;
				stateFadenzugmotor := FADENZUG_MOVE;
			END_IF

			IF MoveAbFadenzugmotorOut1.Error THEN
				stateFadenzugmotor := FADENZUG_ERROR;
			END_IF
			//******************************************************
		ELSIF FadenmotorFreigabe = FALSE THEN
			stateFadenzugmotor := FADENZUG_HALT_ZU_INT;
		END_IF
(* ===========================================================================================		
	Zustand 5: Die Funktion ist gleich wie Zustand 4, aber mithilfe dises Zustands kann den letzte Positionsbefehel unterbrechen 
	und schnell den neue Positionsbefehel aktualisieret und ersetzt werden. *)		
	FADENZUG_MOVE_NEW:

		IF FadenmotorFreigabe = TRUE THEN
			
			IF FadenzugmotorStopp = TRUE THEN
				FadenmotorFreigabe := FALSE;
			END_IF
			
			//*********Positionsführungsgröße berechnen*************
			PRG_PID_Fadenzugmotor();
			IF ILC_EinAus = TRUE AND MasterStart = TRUE THEN
				ILC();
				MoveAbFadenzugmotor2.Position := ILC_Out + GlobaleVariablen.Fadenzugmotor.NcToPlc.ActPos + _u;
			ELSE
				MoveAbFadenzugmotor2.Position := GlobaleVariablen.Fadenzugmotor.NcToPlc.ActPos + _u;
			END_IF
			MoveAbFadenzugmotor2.Velocity := 60000;
			ActBegrenzung_2();
			//******************************************************
			
			MoveAbFadenzugmotor2.Execute := TRUE;
			FadenzugmotorLaeuft := TRUE;
			
			//*********Zustand umschalten***************************
			IF MoveAbFadenzugmotorOut2.Busy OR MoveAbFadenzugmotorOut2.Active THEN
				MoveAbFadenzugmotor2.Execute := FALSE;
				stateFadenzugmotor := FADENZUG_MOVE;
			ELSIF MoveAbFadenzugmotorOut2.Done OR MoveAbFadenzugmotorOut2.CommandAborted THEN
				MoveAbFadenzugmotor2.Execute := FALSE;
				stateFadenzugmotor := FADENZUG_MOVE_NEW;
			ELSIF MoveAbFadenzugmotorOut2.Error THEN
				stateFadenzugmotor := FADENZUG_ERROR;
			END_IF
			//******************************************************
		ELSIF FadenmotorFreigabe = FALSE THEN
			stateFadenzugmotor := FADENZUG_HALT_ZU_INT;
		END_IF
(* ===========================================================================================
   Zustand 7: Anhalten des Fadenzugmotors, im Anschluss Rückkehr in den Ausgangszustand. *)			
	FADENZUG_HALT_ZU_INT:
		MoveAbFadenzugmotor1.Execute := FALSE;
		MoveAbFadenzugmotor2.Execute := FALSE;
		HaltFadenzugmotor.Execute := TRUE;
		IF HaltFadenzugmotorOut.Done THEN
			FadenzugmotorStopp := TRUE;
			FadenmotorFreigabe := FALSE;
			FadenzugmotorLaeuft := FALSE;
			HaltFadenzugmotor.Execute := FALSE;
			stateFadenzugmotor := FADENZUG_INIT;
		ELSIF HaltFadenzugmotorOut.Error OR HaltFadenzugmotorOut.CommandAborted THEN
			HaltFadenzugmotor.Execute := FALSE;
			stateFadenzugmotor := FADENZUG_ERROR;
		END_IF

(* ===========================================================================================
   Zustand 8: Im Falle eines Bausteinfehlers wird überprüft, ob sich die Achse ebenfalls im    
   Fehlerzustand befindet, was einen Achsreset erfordert. Andernfalls werden Bausteinfehler 
   im Zustand Init zurückgesetzt.*)				
	FADENZUG_ERROR:
		MoveAbFadenzugmotor1.Execute := FALSE;
		MoveAbFadenzugmotor2.Execute := FALSE;
		PowerFadenzugmotor.Enable := FALSE;
		FadenmotorFreigabe := FALSE;
		IF Fadenzugmotor.Status.Error THEN
			stateFadenzugmotor := FADENZUG_RESET;	// Reset bei Achsfehler
		ELSE
			stateFadenzugmotor := FADENZUG_INIT;	// Funktionsbausteinfehler erfordert keinen Reset
		END_IF
(* ===========================================================================================
   Zustand 9:  Durchführung des Achsreset im Fehlerfall  *)	
	FADENZUG_RESET:
		MoveAbFadenzugmotor1.Execute := FALSE;
		MoveAbFadenzugmotor2.Execute := FALSE;
		PowerFadenzugmotor.Enable := FALSE;
		ResetFadenzugmotor.Execute := TRUE;
		FadenmotorFreigabe := FALSE;
		IF ResetFadenzugmotor.Done THEN
			FadenzugmotorLaeuft := FALSE;
			stateFadenzugmotor := FADENZUG_INIT;
		ELSIF ResetFadenzugmotorOut.Error THEN
			stateFadenzugmotor := FADENZUG_INIT; (* Falls Reset nicht gelingt, Benutzereingriff erforderlich *)
		END_IF
END_CASE

// Zyklusmäßige Aufrufe
ActPower();		// Aufruf des Funktionsbausteines
ActHalt();
ActRest();
ActMoveAbsolute();

ACTION ActBegrenzung_1:

IF FadenzugmotorAnAus.MoveAbFadenzugmotor1.Position > MaxPosition THEN
	MoveAbFadenzugmotor1.Position := MaxPosition;
	MoveAbFadenzugmotor1.Velocity := 100;
ELSIF FadenzugmotorAnAus.MoveAbFadenzugmotor1.Position < MinPosition THEN
	MoveAbFadenzugmotor1.Position := MinPosition;
	MoveAbFadenzugmotor1.Velocity := 100;
END_IF

IF Fadenzugmotor.NcToPlc.ActPos < MinPosition THEN
	MoveAbFadenzugmotor1.Position := MinPosition;
	MoveAbFadenzugmotor1.Velocity := 100;
	MoveAbFadenzugmotor1.Execute := TRUE;
ELSIF Fadenzugmotor.NcToPlc.ActPos > MaxPosition THEN
	MoveAbFadenzugmotor1.Position := MaxPosition;
	MoveAbFadenzugmotor1.Velocity := 100;
	MoveAbFadenzugmotor1.Execute := TRUE;
END_IF
END_ACTION

ACTION ActBegrenzung_2:
IF MoveAbFadenzugmotor2.Position > MaxPosition THEN
MoveAbFadenzugmotor2.Position := MaxPosition;
MoveAbFadenzugmotor2.Velocity := 100;
ELSIF MoveAbFadenzugmotor2.Position < MinPosition THEN
	MoveAbFadenzugmotor2.Position := MinPosition;
	MoveAbFadenzugmotor2.Velocity := 100;
END_IF

IF Fadenzugmotor.NcToPlc.ActPos < MinPosition THEN
	MoveAbFadenzugmotor2.Position := MinPosition;
	MoveAbFadenzugmotor2.Velocity := 100;
	MoveAbFadenzugmotor2.Execute := TRUE;
ELSIF Fadenzugmotor.NcToPlc.ActPos > MaxPosition THEN
	MoveAbFadenzugmotor2.Position := MaxPosition;
	MoveAbFadenzugmotor2.Velocity := 100;
	MoveAbFadenzugmotor2.Execute := TRUE;
END_IF
END_ACTION

ACTION ActHalt:
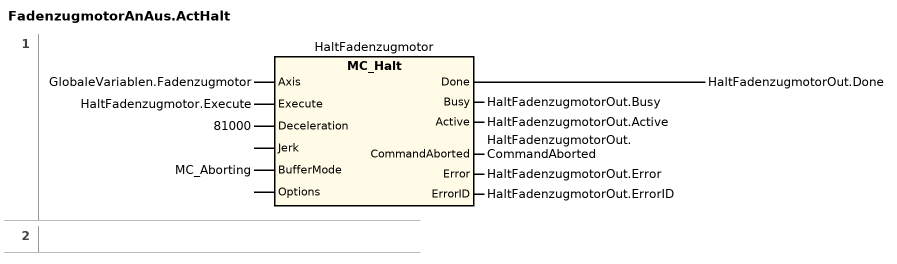
// NETWORK 1
HaltFadenzugmotor(
    Axis := GlobaleVariablen.Fadenzugmotor,
    Execute := HaltFadenzugmotor.Execute,
    Deceleration := 81000,
    BufferMode := MC_Aborting,
    Busy => HaltFadenzugmotorOut.Busy,
    Active => HaltFadenzugmotorOut.Active,
    CommandAborted => HaltFadenzugmotorOut.CommandAborted,
    Error => HaltFadenzugmotorOut.Error,
    ErrorID => HaltFadenzugmotorOut.ErrorID); // MC_Halt
HaltFadenzugmotorOut.Done := HaltFadenzugmotor.Done;

// NETWORK 2
END_ACTION

ACTION ActJog:
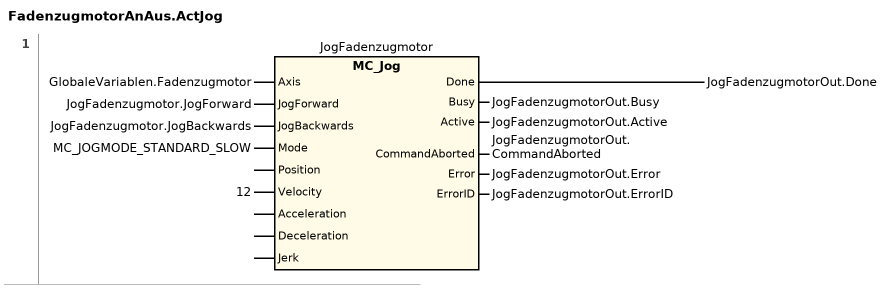
// NETWORK 1
JogFadenzugmotor(
    Axis := GlobaleVariablen.Fadenzugmotor,
    JogForward := JogFadenzugmotor.JogForward,
    JogBackwards := JogFadenzugmotor.JogBackwards,
    Mode := MC_JOGMODE_STANDARD_SLOW,
    Velocity := 12,
    Busy => JogFadenzugmotorOut.Busy,
    Active => JogFadenzugmotorOut.Active,
    CommandAborted => JogFadenzugmotorOut.CommandAborted,
    Error => JogFadenzugmotorOut.Error,
    ErrorID => JogFadenzugmotorOut.ErrorID); // MC_Jog
JogFadenzugmotorOut.Done := JogFadenzugmotor.Done;
END_ACTION

ACTION ActMoveAbsolute:
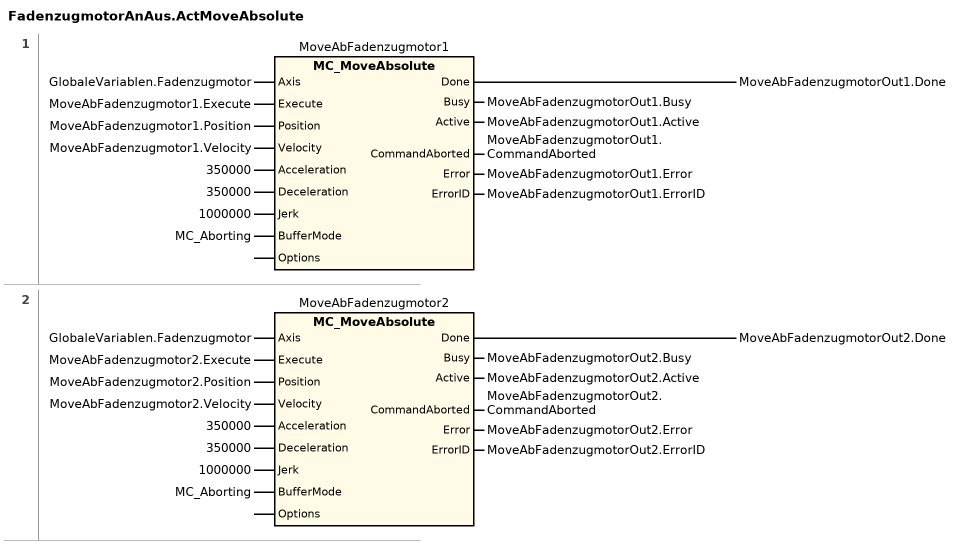
// NETWORK 1
MoveAbFadenzugmotor1(
    Axis := GlobaleVariablen.Fadenzugmotor,
    Execute := MoveAbFadenzugmotor1.Execute,
    Position := MoveAbFadenzugmotor1.Position,
    Velocity := MoveAbFadenzugmotor1.Velocity,
    Acceleration := 350000,
    Deceleration := 350000,
    Jerk := 1000000,
    BufferMode := MC_Aborting,
    Busy => MoveAbFadenzugmotorOut1.Busy,
    Active => MoveAbFadenzugmotorOut1.Active,
    CommandAborted => MoveAbFadenzugmotorOut1.CommandAborted,
    Error => MoveAbFadenzugmotorOut1.Error,
    ErrorID => MoveAbFadenzugmotorOut1.ErrorID); // MC_MoveAbsolute
MoveAbFadenzugmotorOut1.Done := MoveAbFadenzugmotor1.Done;

// NETWORK 2
MoveAbFadenzugmotor2(
    Axis := GlobaleVariablen.Fadenzugmotor,
    Execute := MoveAbFadenzugmotor2.Execute,
    Position := MoveAbFadenzugmotor2.Position,
    Velocity := MoveAbFadenzugmotor2.Velocity,
    Acceleration := 350000,
    Deceleration := 350000,
    Jerk := 1000000,
    BufferMode := MC_Aborting,
    Busy => MoveAbFadenzugmotorOut2.Busy,
    Active => MoveAbFadenzugmotorOut2.Active,
    CommandAborted => MoveAbFadenzugmotorOut2.CommandAborted,
    Error => MoveAbFadenzugmotorOut2.Error,
    ErrorID => MoveAbFadenzugmotorOut2.ErrorID); // MC_MoveAbsolute
MoveAbFadenzugmotorOut2.Done := MoveAbFadenzugmotor2.Done;
END_ACTION

ACTION ActPower:
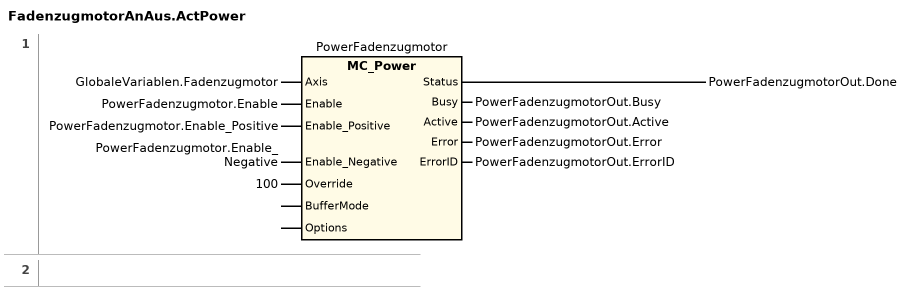
// NETWORK 1
PowerFadenzugmotor(
    Axis := GlobaleVariablen.Fadenzugmotor,
    Enable := PowerFadenzugmotor.Enable,
    Enable_Positive := PowerFadenzugmotor.Enable_Positive,
    Enable_Negative := PowerFadenzugmotor.Enable_Negative,
    Override := 100,
    Busy => PowerFadenzugmotorOut.Busy,
    Active => PowerFadenzugmotorOut.Active,
    Error => PowerFadenzugmotorOut.Error,
    ErrorID => PowerFadenzugmotorOut.ErrorID); // MC_Power
PowerFadenzugmotorOut.Done := PowerFadenzugmotor.Status;

// NETWORK 2
END_ACTION

ACTION ActRest:
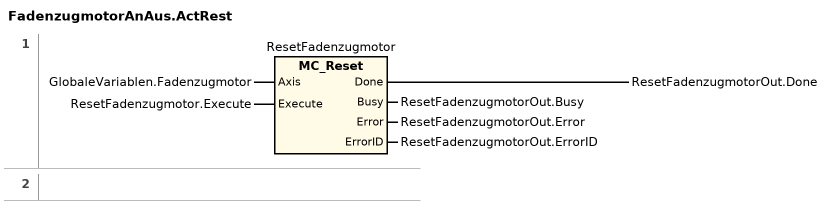
// NETWORK 1
ResetFadenzugmotor(
    Axis := GlobaleVariablen.Fadenzugmotor,
    Execute := ResetFadenzugmotor.Execute,
    Busy => ResetFadenzugmotorOut.Busy,
    Error => ResetFadenzugmotorOut.Error,
    ErrorID => ResetFadenzugmotorOut.ErrorID); // MC_Reset
ResetFadenzugmotorOut.Done := ResetFadenzugmotor.Done;

// NETWORK 2
END_ACTION

END_PROGRAM

// ---- POUs/Regelungsmethode/ADRC-Regler/TrackingDifferentiator.TcPOU
FUNCTION TrackingDifferentiator :LREAL

VAR_INPUT
	expect:LREAL;
END_VAR

v1 := v1 + ADRC_TD_h0 * v2;//跟新最速跟踪状态量x1
v2 := v2 + ADRC_TD_h0 * (-ADRC_TD_r0 * Sign(v1 - expect + (v2 * ABS(v2))/(2 * ADRC_TD_r0)));//跟新最速跟踪状态量微分x2

END_FUNCTION

// ---- POUs/Regelungsmethode/ADRC-Regler/Sign.TcPOU
FUNCTION Sign : LREAL
VAR_INPUT
	Input:LREAL;
END_VAR
VAR
END_VAR

// sign符号函数
IF Input < 0 THEN
	Sign := -1;
ELSIF Input > 0 THEN
	Sign := 1;
ELSE Sign := 0;
END_IF

END_FUNCTION

// ---- POUs/Regelungsmethode/ADRC-Regler/DiscreteTrackingDifferentiator.TcPOU
FUNCTION DiscreteTrackingDifferentiator : LREAL
VAR_INPUT
	expect_ADRC:LREAL;
END_VAR

VAR
	_d:LREAL;
	a0:LREAL;
	_y:LREAL;
	a1:LREAL;
	a2:LREAL;
	_a:LREAL;
    v1_delta: LREAL;//ADRC状态跟踪误差项
	Sy: LREAL;
	Sa: LREAL;
	fhan: LREAL;
END_VAR

v1_delta := v1 - expect_ADRC;//用x1-v(k)替代x1得到离散更新公式

_d := ADRC_TD_r0 * ADRC_TD_h0 * ADRC_TD_h0;//d=r0 * h0^2;
a0 := ADRC_TD_h0 * v2;//a0=h0*v2
_y := v1_delta + a0;//y=x1+a0
a1 := SQRT(_d * (_d + 8.0 * ABS(_y)));//a1=sqrt(d*(d+8*ABS(y))])
a2 := a0 + Sign(_y) * (a1 - _d) / 2.0;//a2=a0+sign(y)*(a1-d)/2;
Sy := (Sign(_y + _d) - Sign(_y - _d)) / 2.0;
_a := (a0 + _y - a2) * Sy + a2;
Sa := (Sign(_a + _d) - Sign(_a - _d)) / 2.0;
fhan := -ADRC_TD_r0 * ((_a / _d) - Sign(_a)) * Sa - ADRC_TD_r0 * Sign(_a);//得到最速微分加速度跟踪量

v1 := v1 + ADRC_TD_h0 * v2;//跟新最速跟踪状态量x1
IF ABS(fhan) <= ADRC_TD_r0 THEN
	v2 := v2 + ADRC_TD_h0 * fhan;//跟新最速跟踪状态量微分x2
END_IF

END_FUNCTION

// ---- POUs/Regelungsmethode/ADRC-Regler/ESO.TcPOU
FUNCTION ESO : LREAL
VAR_INPUT
	_y:LREAL;
END_VAR
VAR
	fe:LREAL;
    fe1:LREAL;
	g1: LREAL;
	g2: LREAL;
	g3: LREAL;
END_VAR

ee := x1_hat - _y;//状态误差

fe := Fal(ee,0.5,ADRC_ESO_h);//非线性函数，提取跟踪状态与当前状态误差
fe1 := Fal(ee,0.25,ADRC_ESO_h);
//g1 := ee;
//g2 := SQRT(ABS(ee)) * Sign(ee);
//g3 := SQRT(SQRT(ABS(ee))) * Sign(ee);

//*************扩展状态量更新**********/
x1_hat := x1_hat + ADRC_ESO_h * (x2_hat - ADRC_ESO_beta01 * ee);
//x1_hat := ADRC_ESO_h * x2_hat - 159 * x1_hat + 160*_y;
x2_hat := x2_hat + ADRC_ESO_h * (x3_hat + b0 * _u - ADRC_ESO_beta02 * fe);
x3_hat := x3_hat + ADRC_ESO_h * (- ADRC_ESO_beta03 * fe1);

END_FUNCTION

// ---- POUs/Regelungsmethode/ADRC-Regler/Fal.TcPOU
FUNCTION Fal : LREAL
VAR_INPUT
	e:LREAL;
	alpha:LREAL;
	delta:LREAL;
END_VAR
VAR
	temp:LREAL;
END_VAR

//原点附近有连线性段的连续幂次函数
IF ABS(e) <= delta THEN
	Fal := e / EXPT(delta, alpha -1);
ELSE
	Fal := EXPT(ABS(e), alpha) * Sign(e);
END_IF
//temp := (Sign(e+delta) - Sign(e-delta)) / 2;
//Fal := e * temp / (EXPT(delta, 1 - alpha)) + EXPT(ABS(e), alpha) * Sign(e) * (1 - temp);

END_FUNCTION

// ---- POUs/Regelungsmethode/PID-Regler/PRG_PID_Fadenzugmotor.TcPOU
PROGRAM PRG_PID_Fadenzugmotor
VAR
	eMode							: E_CTRL_MODE;
	stCTRL_P_PARAMS_Fadenzugmotor					: ST_CTRL_P_PARAMS;
	stCTRL_I_PARAMS_Fadenzugmotor					: ST_CTRL_I_PARAMS;
	stCTRL_D_PARAMS_Fadenzugmotor					: ST_CTRL_D_PARAMS;
	eErrorId						: E_CTRL_ERRORCODES;
	bInit							: BOOL	:= TRUE;
	fManSyncValue					: LREAL;
	bSync							: BOOL;
	bError							: BOOL;
	FB_P_Fadenzugmotor: FB_CTRL_P;
	FB_I_Fadenzugmotor: FB_CTRL_I;
	FB_D_Fadenzugmotor: FB_CTRL_D;
	I_Saturation_Fadenzugmotor: BOOL;
	PID_Regler_Output_Fadenzugmotor: LREAL;
	Fehler_Fadenzugmotor: LREAL;
	Kp: LREAL := 1;
	ADRC_Kp: LREAL := 1;
	Ki: LREAL := 0;
	ADRC_Kd: LREAL := 0.001;
	Kd: LREAL := 0;
	Ti: TIME := T#30S;
	Tv: TIME := T#10MS;
	Td: TIME := T#400MS;
	FB_Vorsteuerung_Fadenzugmotor: FB_CTRL_D;
	stCTRL_Vorsteuerung_PARAMS_Fadenzugmotor: ST_CTRL_D_PARAMS;
	Vorsteuerung_Regler_Out_Fadenzugmotor: LREAL;
	Integral: LREAL;
	I_Halt: BOOL;
	alteKraftfehler: ARRAY[0..9] OF LREAL;
	Differenzial: LREAL;
	x1: LREAL;
	x2: LREAL;
	_d:LREAL:=0;
	a0:LREAL:=0;
	_y:LREAL:=0;
	a1:LREAL:=0;
	a2:LREAL:=0;
	_a:LREAL:=0;
    x1_delta:LREAL:=0;//ADRC状态跟踪误差项
	fh:LREAL:=0;//最速微分加速度跟踪量
END_VAR

IF E_Switch THEN
	IF TD_Switch THEN
		_u_neu := (v1 - x1_hat) * ADRC_Kp + (v2 - x2_hat) * ADRC_Kd ;
	ELSE 
		_u_neu := (Sollkraft - x1_hat) * ADRC_Kp;
	END_IF
	
	_u := (_u_neu - x3_hat) / b0;
	_u := -_u;//Die Richtung der Fadenzugmotor anpassen
ELSE
	IF TD_Switch THEN
		Kraftfehler := v1 - Fadenzugkraft_2;
		Differenzial := v2;
	ELSE
		Kraftfehler := Sollkraft - Fadenzugkraft_2;
		Differenzial := (Kraftfehler - alteKraftfehler[9])/ 0.001;
	END_IF
	
	IF I_Halt = FALSE THEN
		Integral := Integral + Kraftfehler * 0.0001;
	END_IF
	
	PID_Regler_Output_Fadenzugmotor := Kraftfehler * Kp + Integral * Ki + Differenzial * Kd ;
	
	alteKraftfehler[9] := alteKraftfehler[8];
	alteKraftfehler[8] := alteKraftfehler[7];
	alteKraftfehler[7] := alteKraftfehler[6];
	alteKraftfehler[6] := alteKraftfehler[5];
	alteKraftfehler[5] := alteKraftfehler[4];
	alteKraftfehler[4] := alteKraftfehler[3];
	alteKraftfehler[3] := alteKraftfehler[2];
	alteKraftfehler[2] := alteKraftfehler[1];
	alteKraftfehler[1] := alteKraftfehler[0];
	alteKraftfehler[0] := Kraftfehler;
	
	IF PID_Regler_Output_Fadenzugmotor >= 200 THEN 
		PID_Output_After_Saturation_Fadenzugmotor := 200;
	ELSIF PID_Regler_Output_Fadenzugmotor <= -200 THEN 
		PID_Output_After_Saturation_Fadenzugmotor := -200;
	ELSE 
		PID_Output_After_Saturation_Fadenzugmotor := PID_Regler_Output_Fadenzugmotor;
	END_IF
	
	(* Conditional Intrgration *)
	IF Sign(Kraftfehler) = Sign(PID_Regler_Output_Fadenzugmotor) AND PID_Output_After_Saturation_Fadenzugmotor <> PID_Regler_Output_Fadenzugmotor THEN 
		I_Halt := TRUE;
	ELSE
		I_Halt := FALSE;
	END_IF
	
	(* Die Richtung der Fadenzugmotor anpassen *)
	_u := -PID_Output_After_Saturation_Fadenzugmotor;
END_IF

END_PROGRAM

// ---- POUs/Regelungsmethode/IterativeLerningControl/ILC.TcPOU
PROGRAM ILC
VAR
	e_new: LREAL;
	
END_VAR

IF LernenFertig = FALSE THEN
	e_new := GlobaleVariablen.Sollkraft - GlobaleVariablen.Fadenzugkraft_2;
	IF (e_new < (GlobaleVariablen.Sollkraft - 1)) OR (e_new > (GlobaleVariablen.Sollkraft + 1)) THEN
		u_new := u_Old[k] - 0.2 * e_new;
	ELSIF (e_new >= (GlobaleVariablen.Sollkraft - 1)) AND (e_new <= (GlobaleVariablen.Sollkraft + 1)) THEN
		u_new := u_Old[k];
	END_IF
	//PRG_MovingAverage_1();// Moving Average Filter
	
	//Verwendung der "heutigen Daten" als Steuersignal
	ILC_Out := u_new;
	IF ABS(alt_xPunkt) > 180 AND ABS(alt_xPunkt) <= 400 THEN
		IF ILC_Out>0 THEN
			ILC_Out := 0;
		ELSIF ILC_Out < 0 AND  ILC_Out < -2 * e_new THEN
			ILC_Out := -2 * e_new;
		END_IF
	ELSIF ABS(alt_xPunkt) > 400 THEN
		IF ILC_Out>0 AND ILC_Out > - 0.5*e_new THEN
			ILC_Out := - 0.5*e_new;
		ELSIF ILC_Out < 0 AND  ILC_Out < -2 * e_new THEN
			ILC_Out := -2 * e_new;
		END_IF
	END_IF
	
	//"heutige Daten" als "alte Daten" sperchern
	u_Old[k] := ILC_Out;
	e_Old[k] := e_new;
	
	IF ABS(alt_xPunkt) <= 180 THEN
		IF ABS(e_new) > 1 THEN
			LernenFertig := FALSE;
			count := 0;
		ELSE 
			count := count + 1;
		END_IF 
		
		IF count >= 1999 THEN
			LernenFertig := TRUE;
		END_IF
		
	ELSIF ABS(alt_xPunkt) > 180 AND ABS(alt_xPunkt) <= 400 THEN
		IF ABS(e_new) > 2 THEN
			LernenFertig := FALSE;
			count := 0;
		ELSE 
			count := count + 1;
		END_IF 
		
		IF count >= 1999 THEN
			LernenFertig := TRUE;
		END_IF
	ELSIF ABS(alt_xPunkt) > 400 THEN
		IF ABS(e_new) > 4 THEN
			LernenFertig := FALSE;
			count := 0;
		ELSE 
			count := count + 1;
		END_IF 
		
		IF count >= 1999 THEN
			LernenFertig := TRUE;
		END_IF
	END_IF
ELSE
	ILC_Out := u_Old[k];
END_IF

IF ABS(alt_xPunkt) <= 180 THEN
	IF ABS(GlobaleVariablen.Sollkraft - GlobaleVariablen.Fadenzugkraft_2) > 1 THEN
		LernenFertig := FALSE;
	END_IF
ELSIF ABS(alt_xPunkt) > 180 AND ABS(alt_xPunkt) <= 400 THEN
	IF ABS(GlobaleVariablen.Sollkraft - GlobaleVariablen.Fadenzugkraft_2) > 2.3 THEN
		LernenFertig := FALSE;
	END_IF
ELSIF ABS(alt_xPunkt) > 400 THEN
	IF ABS(GlobaleVariablen.Sollkraft - GlobaleVariablen.Fadenzugkraft_2) > 4 THEN
		LernenFertig := FALSE;
	END_IF
END_IF

END_PROGRAM

// ---- POUs/MAIN.TcPOU
(* ===========================================================================================
   Das Hauptprogramm regelt den Gesamtablauf und das Zusammenspiel der Unterprogramme, 
   sodass 
*)

PROGRAM MAIN
VAR
	bErrAck_Button AT %I*:BOOL;
	bErrAck_SAFETY AT %Q*:BOOL;
	
	Timer:LREAL;
	flag:INT;
	Test:BOOL;
END_VAR

// Durchschleifen der Fehler-Quittierung
bErrAck_SAFETY := bErrAck_Button;

// automatisches NOT-AUS laut der Position des Fadenzugmotors
IF Fadenzugmotor.NcToPlc.ActPos < MinPosition + 10 OR Fadenzugmotor.NcToPlc.ActPos > MaxPosition - 10 OR GlobaleVariablen.Fadenzugkraft_2 > 35 THEN
	NOT_AUS := TRUE;
END_IF

//Eine Umdrehung der Masterachse ist ein Zyklus des Textilprozess
IF MasterStart THEN
	Drehzahl := (LREAL_TO_INT(GlobaleVariablen.Master.NcToPlc.ActPos)) MOD 360;
	IF Drehzahl = 0 THEN
		k := 0;
	ELSE
		k := k + 1;
	END_IF
END_IF	

IF Test THEN
	IF Timer >= 10000 THEN
		Timer := 0;
		IF flag = 0 THEN
			flag := 1;
		ELSE
			flag := -flag;
		END_IF
	ELSE
		Timer := Timer + 1;
	END_IF
ELSE
	flag := 0;
END_IF

IF flag = 1 THEN
	Sollkraft := 6;
ELSIF flag = -1 THEN
	Sollkraft := 14;
ELSE
	Sollkraft := 10;
END_IF

IF MasterLaeuft = FALSE AND AbwicklerLaeuft = FALSE AND AufwicklerLaeuft = FALSE THEN
	NOT_AUS := FALSE;
	MasterStopp := FALSE;
	AbwicklerStopp := FALSE;
	AufwicklerStopp := FALSE;
	FadenzugmotorStopp := FALSE;
	FadenmotorRegeln := FALSE;
ELSIF NOT_AUS = TRUE THEN
	MasterStopp := TRUE;
	MasterStart := FALSE;
	FadenmotorRegeln := FALSE;
	AbwicklerStopp := TRUE;
	AufwicklerStopp := TRUE;
	FadenmotorFreigabe := FALSE;
	ILC_EinAus := FALSE;
	Test := FALSE;
	LernenFertig := FALSE;
END_IF


// Status der Achsen am Beginn jedes Zyklus aktualisieren
//GlobaleVariablen.Master();
//GlobaleVariablen.Abwickler();
//GlobaleVariablen.Aufwickler();
//GlobaleVariablen.Fadenzugmotor();

// EL7201-Analogsignal und Positionsabweichung des Ab- und Aufwicklers bearbeiten
//Datenbearbeiten();

// Programmablauf mittels Zustandsautomat
//MasterAnAus();
//AbwicklerAnAus();
//AufwicklerAnAus();
//FadenzugmotorAnAus();

END_PROGRAM

// ---- POUs/Regelungsmethode/IterativeLerningControl/PRG_MovingAverage_1.TcPOU
PROGRAM PRG_MovingAverage_1
VAR
	fActualValue					: LREAL;
	fManSyncValue					: LREAL;
	bSync							: BOOL;
	bHold							: BOOL;

	fOut							: LREAL;
	eMode							: E_CTRL_MODE;
	stCTRL_MOVING_AVERAGE			: ST_CTRL_MOVING_AVERAGE_PARAMS;

	eErrorId						: E_CTRL_ERRORCODES;
	bError							: BOOL;

	(* Filter *)
	arrTable						: ARRAY[1..10] OF FLOAT;
	fbCTRL_MOVING_AVERAGE			: FB_CTRL_MOVING_AVERAGE;

	bInit							: BOOL		:= TRUE;
END_VAR

IF bInit THEN
	(* init parameter struct *)
	stCTRL_MOVING_AVERAGE.tCtrlCycleTime		:= T#10MS;
	stCTRL_MOVING_AVERAGE.tTaskCycleTime		:= T#10MS;
	stCTRL_MOVING_AVERAGE.nSamplesToFilter		:= 10;

	(* set the mode to ACTIVE --> normal operation *)
	eMode := eCTRL_MODE_ACTIVE;

	(* reset the init flag *)
	bInit := FALSE;
END_IF

(* set the addresses *)
stCTRL_MOVING_AVERAGE.pWorkArray_ADR		:= ADR(arrTable);
stCTRL_MOVING_AVERAGE.nWorkArray_SIZEOF		:= SIZEOF(arrTable);

(* call the filter *)
fbCTRL_MOVING_AVERAGE	(	fIn				:= u_new,
							fManSyncValue	:= fManSyncValue,
							bSync			:= bSync,
							eMode			:= eMode,
							stParams		:= stCTRL_MOVING_AVERAGE,
							bHold			:= bHold,
							fOut			=> ILC_F_Out,
							eErrorId		=> eErrorId,
							bError			=> bError
							);

END_PROGRAM

// ---- POUs/Regelungsmethode/KraftwerteBearbeiten/PRG_MovingAverage.TcPOU
PROGRAM PRG_MovingAverage
VAR
	fActualValue					: LREAL;
	fManSyncValue					: LREAL;
	bSync							: BOOL;
	bHold							: BOOL;

	fOut							: LREAL;
	eMode							: E_CTRL_MODE;
	stCTRL_MOVING_AVERAGE			: ST_CTRL_MOVING_AVERAGE_PARAMS;

	eErrorId						: E_CTRL_ERRORCODES;
	bError							: BOOL;

	(* Filter *)
	arrTable						: ARRAY[1..10] OF FLOAT;
	fbCTRL_MOVING_AVERAGE			: FB_CTRL_MOVING_AVERAGE;

	bInit							: BOOL		:= TRUE;
END_VAR

IF bInit THEN
	(* init parameter struct *)
	stCTRL_MOVING_AVERAGE.tCtrlCycleTime		:= T#10ms;
	stCTRL_MOVING_AVERAGE.tTaskCycleTime		:= T#10ms;
	stCTRL_MOVING_AVERAGE.nSamplesToFilter		:= 10;

	(* set the mode to ACTIVE --> normal operation *)
	eMode := eCTRL_MODE_ACTIVE;

	(* reset the init flag *)
	bInit := FALSE;
END_IF

(* set the addresses *)
stCTRL_MOVING_AVERAGE.pWorkArray_ADR		:= ADR(arrTable);
stCTRL_MOVING_AVERAGE.nWorkArray_SIZEOF		:= SIZEOF(arrTable);

(* call the filter *)
fbCTRL_MOVING_AVERAGE	(	fIn				:= GlobaleVariablen.iAnalogSamplesAverageValue_2,
							fManSyncValue	:= fManSyncValue,
							bSync			:= bSync,
							eMode			:= eMode,
							stParams		:= stCTRL_MOVING_AVERAGE,
							bHold			:= bHold,
							fOut			=> GlobaleVariablen.iAnalogSamplesAverageValue_2,
							eErrorId		=> eErrorId,
							bError			=> bError
							);

END_PROGRAM

// ---- POUs/Regelungsmethode/PID-Regler/PRG_PID_Abwickler.TcPOU
PROGRAM PRG_PID_Abwickler
VAR
	Fehler_Abwickler: LREAL;
	eMode							: E_CTRL_MODE;
	stCTRL_P_PARAMS_Abwickler					: ST_CTRL_P_PARAMS;
	stCTRL_I_PARAMS_Abwickler					: ST_CTRL_I_PARAMS;
	stCTRL_D_PARAMS_Abwickler					: ST_CTRL_D_PARAMS;
	eErrorId						: E_CTRL_ERRORCODES;
	bInit							: BOOL	:= TRUE;
	fManSyncValue					: LREAL;
	bSync							: BOOL;
	bError							: BOOL;
	FB_P_Abwickler: FB_CTRL_P;
	FB_I_Abwickler: FB_CTRL_I;
	FB_D_Abwickler: FB_CTRL_D;
	I_Saturation_Abwickler: BOOL;
	PID_Regler_Output_Abwickler: LREAL;
END_VAR

Fehler_Abwickler := Referenzposition - Fadenzugmotor.NcToPlc.ActPos;

IF bInit THEN
	(* init parameter struct *)
	stCTRL_P_PARAMS_Abwickler.tCtrlCycleTime := T#1MS;
	stCTRL_P_PARAMS_Abwickler.tTaskCycleTime := T#1MS;
	stCTRL_P_PARAMS_Abwickler.fKp			 := 1;
	
	stCTRL_I_PARAMS_Abwickler.tCtrlCycleTime := T#100MS;
	stCTRL_I_PARAMS_Abwickler.tTaskCycleTime := T#100MS;
	stCTRL_I_PARAMS_Abwickler.tTi			 := T#50MS;
	stCTRL_I_PARAMS_Abwickler.fOutMaxLimit	 := 40;
	stCTRL_I_PARAMS_Abwickler.fOutMinLimit	 := -40;
	
	stCTRL_D_PARAMS_Abwickler.tCtrlCycleTime := T#1MS;
	stCTRL_D_PARAMS_Abwickler.tTaskCycleTime := T#1MS;
	stCTRL_D_PARAMS_Abwickler.tTv			 := T#3S;
	stCTRL_D_PARAMS_Abwickler.tTd			 := T#10MS;
	stCTRL_D_PARAMS_Abwickler.fOutMaxLimit	 :=  40;
	stCTRL_D_PARAMS_Abwickler.fOutMinLimit	 := -40;

	(* reset the init flag *)
	bInit	:= FALSE;
END_IF	 

(* ein idealer PID-Regler in der Summendarstellung der Parameter *)
FB_PID_Regler_Abwickler();
PID_Regler_Output_Abwickler := P_Regler_Out_Abwickler + I_Regler_Out_Abwickler + D_Regler_Out_Abwickler;	 
//PID_Regler_Output_Abwickler := I_Regler_Out_Abwickler;

IF PID_Regler_Output_Abwickler > 40 THEN 
	PID_Output_After_Saturation_Abwickler := 40;
ELSIF PID_Regler_Output_Abwickler < -40 THEN 
	PID_Output_After_Saturation_Abwickler := -40;
ELSE 
	PID_Output_After_Saturation_Abwickler := PID_Regler_Output_Abwickler;
END_IF	

(* Conditional Intrgration *)
IF Sign(Fehler_Abwickler) = Sign(PID_Regler_Output_Abwickler) AND PID_Output_After_Saturation_Abwickler <> PID_Regler_Output_Abwickler THEN 
	FB_I_Abwickler.bHold := TRUE;
ELSE FB_I_Abwickler.bHold := FALSE;
END_IF

(* Die Richtung der Tänzerregelung anpassen *)
PID_Output_After_Saturation_Abwickler := -PID_Output_After_Saturation_Abwickler;

ACTION FB_PID_Regler_Abwickler:
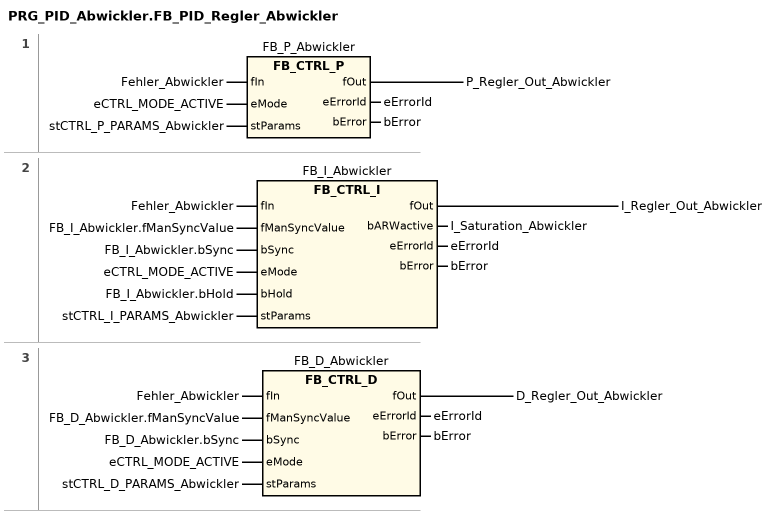
// NETWORK 1
FB_P_Abwickler(
    fIn := Fehler_Abwickler,
    eMode := eCTRL_MODE_ACTIVE,
    stParams := stCTRL_P_PARAMS_Abwickler,
    eErrorId => eErrorId,
    bError => bError); // FB_CTRL_P
P_Regler_Out_Abwickler := FB_P_Abwickler.fOut;

// NETWORK 2
FB_I_Abwickler(
    fIn := Fehler_Abwickler,
    fManSyncValue := FB_I_Abwickler.fManSyncValue,
    bSync := FB_I_Abwickler.bSync,
    eMode := eCTRL_MODE_ACTIVE,
    bHold := FB_I_Abwickler.bHold,
    stParams := stCTRL_I_PARAMS_Abwickler,
    bARWactive => I_Saturation_Abwickler,
    eErrorId => eErrorId,
    bError => bError); // FB_CTRL_I
I_Regler_Out_Abwickler := FB_I_Abwickler.fOut;

// NETWORK 3
FB_D_Abwickler(
    fIn := Fehler_Abwickler,
    fManSyncValue := FB_D_Abwickler.fManSyncValue,
    bSync := FB_D_Abwickler.bSync,
    eMode := eCTRL_MODE_ACTIVE,
    stParams := stCTRL_D_PARAMS_Abwickler,
    eErrorId => eErrorId,
    bError => bError); // FB_CTRL_D
D_Regler_Out_Abwickler := FB_D_Abwickler.fOut;
END_ACTION

END_PROGRAM

// ---- GlobalTextList.TcGTLO
TEXTLIST GlobalTextList
  643 = '%.0f'
  805 = '%.f'
  41 = '%f'
  688 = 'Bereit'
  153 = 'GlobaleVariablen.Position'
  424 = 'GlobaleVariablen.Sollposition'
  132 = 'Motorfreigabe'
  855 = 'Übergrenzung'
END_TEXTLIST
